LIN {X 0,Y 525.332,Z 477.044,A -85,B 0,C 180,E1 -4784.626,E2 -4784.626} C_VEL
LIN {X 0,Y 525.652,Z 463.482,A -85,B 0,C 180,E1 -4785.311,E2 -4785.311} C_VEL
LIN {X 0,Y 525.936,Z 448.87,A -85,B 0,C 180,E1 -4785.862,E2 -4785.862} C_VEL
LIN {X 0,Y 526.206,Z 434.89,A -85,B 0,C 180,E1 -4786.225,E2 -4786.225} C_VEL
LIN {X 0,Y 526.347,Z 409.491,A -85,B 0,C 180,E1 -4786.608,E2 -4786.608} C_VEL
LIN {X 0,Y 526.914,Z 305.92,A -85,B 0,C 180,E1 -4788.059,E2 -4788.059} C_VEL
LIN {X 0,Y 525.207,Z 295.454,A -85,B 0,C 180,E1 -4788.29,E2 -4788.29} C_VEL
LIN {X 0,Y 525.997,Z 269.747,A -85,B 0,C 180,E1 -4791.557,E2 -4791.557} C_VEL
LIN {X 0,Y 526.502,Z 253.973,A -85,B 0,C 180,E1 -4793.606,E2 -4793.606} C_VEL
LIN {X 0,Y 524.008,Z 242.955,A -85,B 0,C 180,E1 -4795.243,E2 -4795.243} C_VEL
LIN {X 0,Y 523.969,Z 242.84,A -85,B 0,C 180,E1 -4797.998,E2 -4797.998} C_VEL
LIN {X 0,Y 523.943,Z 242.842,A -85,B 0,C 180,E1 -4800.854,E2 -4800.854} C_VEL
LIN {X 0,Y 523.957,Z 242.841,A -85,B 0,C 180,E1 -4803.734,E2 -4803.734} C_VEL
LIN {X 0,Y 523.9,Z 242.841,A -85,B 0,C 180,E1 -4806.401,E2 -4806.401} C_VEL
LIN {X 0,Y 523.917,Z 242.846,A -85,B 0,C 180,E1 -4809.084,E2 -4809.084} C_VEL
LIN {X 0,Y 523.952,Z 242.844,A -85,B 0,C 180,E1 -4812.118,E2 -4812.118} C_VEL
LIN {X 0,Y 523.951,Z 242.838,A -85,B 0,C 180,E1 -4815.308,E2 -4815.308} C_VEL
LIN {X 0,Y 523.957,Z 242.838,A -85,B 0,C 180,E1 -4818.689,E2 -4818.689} C_VEL
LIN {X 0,Y 523.912,Z 242.85,A -85,B 0,C 180,E1 -4821.898,E2 -4821.898} C_VEL
LIN {X 0,Y 523.933,Z 242.839,A -85,B 0,C 180,E1 -4824.908,E2 -4824.908} C_VEL
LIN {X 0,Y 523.937,Z 242.845,A -85,B 0,C 180,E1 -4827.678,E2 -4827.678} C_VEL
LIN {X 0,Y 523.957,Z 242.834,A -85,B 0,C 180,E1 -4830.674,E2 -4830.674} C_VEL
LIN {X 0,Y 523.969,Z 242.843,A -85,B 0,C 180,E1 -4833.728,E2 -4833.728} C_VEL
LIN {X 0,Y 523.93,Z 242.846,A -85,B 0,C 180,E1 -4836.271,E2 -4836.271} C_VEL
LIN {X 0,Y 523.939,Z 242.84,A -85,B 0,C 180,E1 -4838.767,E2 -4838.767} C_VEL
LIN {X 0,Y 523.947,Z 242.841,A -85,B 0,C 180,E1 -4841.221,E2 -4841.221} C_VEL
LIN {X 0,Y 523.934,Z 242.847,A -85,B 0,C 180,E1 -4843.639,E2 -4843.639} C_VEL
LIN {X 0,Y 523.934,Z 242.846,A -85,B 0,C 180,E1 -4846.028,E2 -4846.028} C_VEL
LIN {X 0,Y 524.005,Z 242.832,A -85,B 0,C 180,E1 -4848.394,E2 -4848.394} C_VEL
LIN {X 0,Y 523.999,Z 242.84,A -85,B 0,C 180,E1 -4851.516,E2 -4851.516} C_VEL
LIN {X 0,Y 524.077,Z 242.824,A -85,B 0,C 180,E1 -4854.614,E2 -4854.614} C_VEL
LIN {X 0,Y 524.105,Z 242.826,A -85,B 0,C 180,E1 -4857.695,E2 -4857.695} C_VEL
LIN {X 0,Y 524.118,Z 242.819,A -85,B 0,C 180,E1 -4860.769,E2 -4860.769} C_VEL
LIN {X 0,Y 524.068,Z 242.825,A -85,B 0,C 180,E1 -4863.075,E2 -4863.075} C_VEL
LIN {X 0,Y 524.04,Z 242.827,A -85,B 0,C 180,E1 -4866.159,E2 -4866.159} C_VEL
LIN {X 0,Y 523.994,Z 242.841,A -85,B 0,C 180,E1 -4869.262,E2 -4869.262} C_VEL
LIN {X 0,Y 523.996,Z 242.836,A -85,B 0,C 180,E1 -4871.74,E2 -4871.74} C_VEL
LIN {X 0,Y 523.987,Z 242.84,A -85,B 0,C 180,E1 -4875.053,E2 -4875.053} C_VEL
LIN {X 0,Y 523.959,Z 242.84,A -85,B 0,C 180,E1 -4877.97,E2 -4877.97} C_VEL
LIN {X 0,Y 523.967,Z 242.836,A -85,B 0,C 180,E1 -4880.411,E2 -4880.411} C_VEL
LIN {X 0,Y 523.912,Z 242.85,A -85,B 0,C 180,E1 -4882.894,E2 -4882.894} C_VEL
LIN {X 0,Y 523.948,Z 242.845,A -85,B 0,C 180,E1 -4885.419,E2 -4885.419} C_VEL
LIN {X 0,Y 523.966,Z 242.833,A -85,B 0,C 180,E1 -4888,E2 -4888} C_VEL
LIN {X 0,Y 523.944,Z 242.843,A -85,B 0,C 180,E1 -4890.856,E2 -4890.856} C_VEL
LIN {X 0,Y 523.958,Z 242.837,A -85,B 0,C 180,E1 -4893.736,E2 -4893.736} C_VEL
LIN {X 0,Y 523.92,Z 242.843,A -85,B 0,C 180,E1 -4896.405,E2 -4896.405} C_VEL
LIN {X 0,Y 523.921,Z 242.845,A -85,B 0,C 180,E1 -4899.085,E2 -4899.085} C_VEL
LIN {X 0,Y 523.952,Z 242.841,A -85,B 0,C 180,E1 -4902.12,E2 -4902.12} C_VEL
LIN {X 0,Y 523.955,Z 242.843,A -85,B 0,C 180,E1 -4905.309,E2 -4905.309} C_VEL
LIN {X 0,Y 523.923,Z 242.847,A -85,B 0,C 180,E1 -4906.918,E2 -4906.918} C_VEL
LIN {X 0,Y 523.256,Z 242.926,A -85,B 0,C 180,E1 -4907.56,E2 -4907.56} C_VEL
LIN {X 0,Y 520.412,Z 243.286,A -85,B 0,C 180,E1 -4908.601,E2 -4908.601} C_VEL
LIN {X 0,Y 518.006,Z 243.59,A -85,B 0,C 180,E1 -4909.44,E2 -4909.44} C_VEL
LIN {X 0,Y 516.968,Z 243.716,A -85,B 0,C 180,E1 -4910.088,E2 -4910.088} C_VEL
LIN {X 0,Y 516.881,Z 243.723,A -85,B 0,C 180,E1 -4910.307,E2 -4910.307} C_VEL
LIN {X 0,Y 516.878,Z 243.724,A -85,B 0,C 180,E1 -4913.344,E2 -4913.344} C_VEL
LIN {X 0,Y 516.886,Z 243.716,A -85,B 0,C 180,E1 -4916.12,E2 -4916.12} C_VEL
LIN {X 0,Y 516.892,Z 243.717,A -85,B 0,C 180,E1 -4918.937,E2 -4918.937} C_VEL
LIN {X 0,Y 516.943,Z 243.918,A -85,B 0,C 180,E1 -4921.799,E2 -4921.799} C_VEL
LIN {X 0,Y 519.069,Z 253.792,A -85,B 0,C 180,E1 -4923.461,E2 -4923.461} C_VEL
LIN {X 0,Y 519.119,Z 260.818,A -85,B 0,C 180,E1 -4924.543,E2 -4924.543} C_VEL
LIN {X 0,Y 518.393,Z 281.839,A -85,B 0,C 180,E1 -4927.691,E2 -4927.691} C_VEL
LIN {X 0,Y 517.797,Z 304.258,A -85,B 0,C 180,E1 -4930.989,E2 -4930.989} C_VEL
LIN {X 0,Y 517.551,Z 314.996,A -85,B 0,C 180,E1 -4932.528,E2 -4932.528} C_VEL
LIN {X 0,Y 519.391,Z 327.308,A -85,B 0,C 180,E1 -4932.783,E2 -4932.783} C_VEL
LIN {X 0,Y 519.012,Z 424.803,A -85,B 0,C 180,E1 -4934.123,E2 -4934.123} C_VEL
LIN {X 0,Y 518.798,Z 437.066,A -85,B 0,C 180,E1 -4934.432,E2 -4934.432} C_VEL
LIN {X 0,Y 518.519,Z 450.121,A -85,B 0,C 180,E1 -4934.926,E2 -4934.926} C_VEL
LIN {X 0,Y 518.167,Z 462.487,A -85,B 0,C 180,E1 -4935.569,E2 -4935.569} C_VEL
LIN {X 0,Y 517.756,Z 474.085,A -85,B 0,C 180,E1 -4936.359,E2 -4936.359} C_VEL
LIN {X 0,Y 517.433,Z 484.503,A -85,B 0,C 180,E1 -4937.249,E2 -4937.249} C_VEL
LIN {X 0,Y 517.067,Z 493.894,A -85,B 0,C 180,E1 -4938.236,E2 -4938.236} C_VEL
LIN {X 0,Y 516.846,Z 502.93,A -85,B 0,C 180,E1 -4939.422,E2 -4939.422} C_VEL
LIN {X 0,Y 516.651,Z 510.21,A -85,B 0,C 180,E1 -4940.605,E2 -4940.605} C_VEL
LIN {X 0,Y 516.474,Z 516.049,A -85,B 0,C 180,E1 -4941.786,E2 -4941.786} C_VEL
LIN {X 0,Y 516.398,Z 520.658,A -85,B 0,C 180,E1 -4942.964,E2 -4942.964} C_VEL
LIN {X 0,Y 516.311,Z 523.127,A -85,B 0,C 180,E1 -4943.748,E2 -4943.748} C_VEL
LIN {X 0,Y 516.318,Z 525.122,A -85,B 0,C 180,E1 -4944.532,E2 -4944.532} C_VEL
LIN {X 0,Y 516.227,Z 526.71,A -85,B 0,C 180,E1 -4945.315,E2 -4945.315} C_VEL
LIN {X 0,Y 516.325,Z 527.898,A -85,B 0,C 180,E1 -4946.098,E2 -4946.098} C_VEL
LIN {X 0,Y 516.26,Z 529.038,A -85,B 0,C 180,E1 -4947.659,E2 -4947.659} C_VEL
LIN {X 0,Y 516.161,Z 528.663,A -85,B 0,C 180,E1 -4949.22,E2 -4949.22} C_VEL
LIN {X 0,Y 516.162,Z 527.89,A -85,B 0,C 180,E1 -4950,E2 -4950} C_VEL
LIN {X 0,Y 516.222,Z 525.112,A -85,B 0,C 180,E1 -4951.56,E2 -4951.56} C_VEL
LIN {X 0,Y 516.347,Z 521.938,A -85,B 0,C 180,E1 -4952.73,E2 -4952.73} C_VEL
LIN {X 0,Y 516.43,Z 517.732,A -85,B 0,C 180,E1 -4953.902,E2 -4953.902} C_VEL
LIN {X 0,Y 516.636,Z 512.373,A -85,B 0,C 180,E1 -4955.073,E2 -4955.073} C_VEL
LIN {X 0,Y 516.742,Z 505.703,A -85,B 0,C 180,E1 -4956.246,E2 -4956.246} C_VEL
LIN {X 0,Y 517,Z 497.426,A -85,B 0,C 180,E1 -4957.42,E2 -4957.42} C_VEL
LIN {X 0,Y 517.34,Z 488.918,A -85,B 0,C 180,E1 -4958.397,E2 -4958.397} C_VEL
LIN {X 0,Y 517.677,Z 478.474,A -85,B 0,C 180,E1 -4959.376,E2 -4959.376} C_VEL
LIN {X 0,Y 517.974,Z 468.125,A -85,B 0,C 180,E1 -4960.159,E2 -4960.159} C_VEL
LIN {X 0,Y 518.32,Z 456.727,A -85,B 0,C 180,E1 -4960.844,E2 -4960.844} C_VEL
LIN {X 0,Y 518.643,Z 443.643,A -85,B 0,C 180,E1 -4961.43,E2 -4961.43} C_VEL
LIN {X 0,Y 518.865,Z 430.369,A -85,B 0,C 180,E1 -4961.846,E2 -4961.846} C_VEL
LIN {X 0,Y 519.002,Z 417.033,A -85,B 0,C 180,E1 -4962.091,E2 -4962.091} C_VEL
LIN {X 0,Y 519.312,Z 325.809,A -85,B 0,C 180,E1 -4963.329,E2 -4963.329} C_VEL
LIN {X 0,Y 517.579,Z 315.248,A -85,B 0,C 180,E1 -4963.546,E2 -4963.546} C_VEL
LIN {X 0,Y 517.655,Z 309.433,A -85,B 0,C 180,E1 -4964.345,E2 -4964.345} C_VEL
LIN {X 0,Y 518.24,Z 287.488,A -85,B 0,C 180,E1 -4967.562,E2 -4967.562} C_VEL
LIN {X 0,Y 518.798,Z 268.307,A -85,B 0,C 180,E1 -4970.415,E2 -4970.415} C_VEL
LIN {X 0,Y 519.199,Z 254.521,A -85,B 0,C 180,E1 -4972.493,E2 -4972.493} C_VEL
LIN {X 0,Y 516.928,Z 243.789,A -85,B 0,C 180,E1 -4974.295,E2 -4974.295} C_VEL
LIN {X 0,Y 516.926,Z 243.707,A -85,B 0,C 180,E1 -4976.657,E2 -4976.657} C_VEL
LIN {X 0,Y 516.913,Z 243.716,A -85,B 0,C 180,E1 -4979.523,E2 -4979.523} C_VEL
LIN {X 0,Y 516.899,Z 243.718,A -85,B 0,C 180,E1 -4982.543,E2 -4982.543} C_VEL
LIN {X 0,Y 516.867,Z 243.726,A -85,B 0,C 180,E1 -4985.329,E2 -4985.329} C_VEL
LIN {X 0,Y 516.88,Z 243.721,A -85,B 0,C 180,E1 -4987.942,E2 -4987.942} C_VEL
LIN {X 0,Y 516.885,Z 243.721,A -85,B 0,C 180,E1 -4990.741,E2 -4990.741} C_VEL
LIN {X 0,Y 516.905,Z 243.721,A -85,B 0,C 180,E1 -4992.828,E2 -4992.828} C_VEL
LIN {X 0,Y 516.922,Z 243.718,A -85,B 0,C 180,E1 -4995.009,E2 -4995.009} C_VEL
LIN {X 0,Y 516.913,Z 243.717,A -85,B 0,C 180,E1 -4998.398,E2 -4998.398} C_VEL
LIN {X 0,Y 516.881,Z 243.726,A -85,B 0,C 180,E1 -5001.283,E2 -5001.283} C_VEL
LIN {X 0,Y 516.888,Z 243.719,A -85,B 0,C 180,E1 -5004.22,E2 -5004.22} C_VEL
LIN {X 0,Y 516.894,Z 243.718,A -85,B 0,C 180,E1 -5007.052,E2 -5007.052} C_VEL
LIN {X 0,Y 516.897,Z 243.719,A -85,B 0,C 180,E1 -5009.796,E2 -5009.796} C_VEL
LIN {X 0,Y 516.924,Z 243.715,A -85,B 0,C 180,E1 -5012.467,E2 -5012.467} C_VEL
LIN {X 0,Y 516.906,Z 243.72,A -85,B 0,C 180,E1 -5015.071,E2 -5015.071} C_VEL
LIN {X 0,Y 516.864,Z 243.723,A -85,B 0,C 180,E1 -5017.621,E2 -5017.621} C_VEL
LIN {X 0,Y 516.927,Z 243.714,A -85,B 0,C 180,E1 -5020.129,E2 -5020.129} C_VEL
LIN {X 0,Y 516.925,Z 243.721,A -85,B 0,C 180,E1 -5022.596,E2 -5022.596} C_VEL
LIN {X 0,Y 516.935,Z 243.716,A -85,B 0,C 180,E1 -5025.03,E2 -5025.03} C_VEL
LIN {X 0,Y 516.958,Z 243.714,A -85,B 0,C 180,E1 -5028.233,E2 -5028.233} C_VEL
LIN {X 0,Y 516.963,Z 243.71,A -85,B 0,C 180,E1 -5031.399,E2 -5031.399} C_VEL
LIN {X 0,Y 517.003,Z 243.705,A -85,B 0,C 180,E1 -5033.756,E2 -5033.756} C_VEL
LIN {X 0,Y 517.077,Z 243.696,A -85,B 0,C 180,E1 -5037.663,E2 -5037.663} C_VEL
LIN {X 0,Y 517.088,Z 243.697,A -85,B 0,C 180,E1 -5040.779,E2 -5040.779} C_VEL
LIN {X 0,Y 517.008,Z 243.705,A -85,B 0,C 180,E1 -5043.117,E2 -5043.117} C_VEL
LIN {X 0,Y 517.003,Z 243.709,A -85,B 0,C 180,E1 -5046.243,E2 -5046.243} C_VEL
LIN {X 0,Y 516.948,Z 243.712,A -85,B 0,C 180,E1 -5049.389,E2 -5049.389} C_VEL
LIN {X 0,Y 516.944,Z 243.712,A -85,B 0,C 180,E1 -5051.807,E2 -5051.807} C_VEL
LIN {X 0,Y 516.936,Z 243.712,A -85,B 0,C 180,E1 -5055.146,E2 -5055.146} C_VEL
LIN {X 0,Y 516.918,Z 243.724,A -85,B 0,C 180,E1 -5058.222,E2 -5058.222} C_VEL
LIN {X 0,Y 516.905,Z 243.717,A -85,B 0,C 180,E1 -5060.702,E2 -5060.702} C_VEL
LIN {X 0,Y 516.904,Z 243.724,A -85,B 0,C 180,E1 -5064.072,E2 -5064.072} C_VEL
LIN {X 0,Y 516.92,Z 243.717,A -85,B 0,C 180,E1 -5066.658,E2 -5066.658} C_VEL
LIN {X 0,Y 516.918,Z 243.715,A -85,B 0,C 180,E1 -5069.527,E2 -5069.527} C_VEL
LIN {X 0,Y 516.894,Z 243.72,A -85,B 0,C 180,E1 -5072.545,E2 -5072.545} C_VEL
LIN {X 0,Y 516.877,Z 243.722,A -85,B 0,C 180,E1 -5075.333,E2 -5075.333} C_VEL
LIN {X 0,Y 516.877,Z 243.725,A -85,B 0,C 180,E1 -5077.944,E2 -5077.944} C_VEL
LIN {X 0,Y 516.881,Z 243.72,A -85,B 0,C 180,E1 -5080.742,E2 -5080.742} C_VEL
LIN {X 0,Y 516.879,Z 243.718,A -85,B 0,C 180,E1 -5082.832,E2 -5082.832} C_VEL
LIN {X 0,Y 516.918,Z 243.717,A -85,B 0,C 180,E1 -5085.011,E2 -5085.011} C_VEL
LIN {X 0,Y 516.912,Z 243.705,A -85,B 0,C 180,E1 -5088.399,E2 -5088.399} C_VEL
LIN {X 0,Y 516.877,Z 243.725,A -85,B 0,C 180,E1 -5091.285,E2 -5091.285} C_VEL
LIN {X 0,Y 516.868,Z 243.716,A -85,B 0,C 180,E1 -5094.22,E2 -5094.22} C_VEL
LIN {X 0,Y 516.894,Z 243.723,A -85,B 0,C 180,E1 -5097.054,E2 -5097.054} C_VEL
LIN {X 0,Y 516.891,Z 243.726,A -85,B 0,C 180,E1 -5099.797,E2 -5099.797} C_VEL
LIN {X 0,Y 516.927,Z 243.719,A -85,B 0,C 180,E1 -5102.468,E2 -5102.468} C_VEL
LIN {X 0,Y 516.958,Z 243.855,A -85,B 0,C 180,E1 -5104.537,E2 -5104.537} C_VEL
LIN {X 0,Y 519.629,Z 255.55,A -85,B 0,C 180,E1 -5106.274,E2 -5106.274} C_VEL
LIN {X 0,Y 519.014,Z 274.477,A -85,B 0,C 180,E1 -5108.761,E2 -5108.761} C_VEL
LIN {X 0,Y 518.331,Z 295.82,A -85,B 0,C 180,E1 -5111.495,E2 -5111.495} C_VEL
LIN {X 0,Y 520.162,Z 307.48,A -85,B 0,C 180,E1 -5111.741,E2 -5111.741} C_VEL
LIN {X 0,Y 519.337,Z 432.731,A -85,B 0,C 180,E1 -5113.537,E2 -5113.537} C_VEL
LIN {X 0,Y 519.113,Z 447.385,A -85,B 0,C 180,E1 -5113.905,E2 -5113.905} C_VEL
LIN {X 0,Y 518.835,Z 460.485,A -85,B 0,C 180,E1 -5114.382,E2 -5114.382} C_VEL
LIN {X 0,Y 518.488,Z 472.87,A -85,B 0,C 180,E1 -5114.976,E2 -5114.976} C_VEL
LIN {X 0,Y 518.09,Z 485.849,A -85,B 0,C 180,E1 -5115.767,E2 -5115.767} C_VEL
LIN {X 0,Y 517.703,Z 497.626,A -85,B 0,C 180,E1 -5116.657,E2 -5116.657} C_VEL
LIN {X 0,Y 517.381,Z 508.456,A -85,B 0,C 180,E1 -5117.652,E2 -5117.652} C_VEL
LIN {X 0,Y 517.067,Z 519.064,A -85,B 0,C 180,E1 -5118.832,E2 -5118.832} C_VEL
LIN {X 0,Y 516.798,Z 527.848,A -85,B 0,C 180,E1 -5120.015,E2 -5120.015} C_VEL
LIN {X 0,Y 516.579,Z 536.259,A -85,B 0,C 180,E1 -5121.393,E2 -5121.393} C_VEL
LIN {X 0,Y 516.445,Z 542.107,A -85,B 0,C 180,E1 -5122.572,E2 -5122.572} C_VEL
LIN {X 0,Y 516.371,Z 546.91,A -85,B 0,C 180,E1 -5123.749,E2 -5123.749} C_VEL
LIN {X 0,Y 516.305,Z 550.799,A -85,B 0,C 180,E1 -5124.924,E2 -5124.924} C_VEL
LIN {X 0,Y 516.324,Z 553.783,A -85,B 0,C 180,E1 -5126.098,E2 -5126.098} C_VEL
LIN {X 0,Y 516.259,Z 556.518,A -85,B 0,C 180,E1 -5127.659,E2 -5127.659} C_VEL
LIN {X 0,Y 516.157,Z 557.872,A -85,B 0,C 180,E1 -5129.22,E2 -5129.22} C_VEL
LIN {X 0,Y 516.157,Z 557.873,A -85,B 0,C 180,E1 -5130.78,E2 -5130.78} C_VEL
LIN {X 0,Y 516.259,Z 556.521,A -85,B 0,C 180,E1 -5132.341,E2 -5132.341} C_VEL
LIN {X 0,Y 516.324,Z 553.788,A -85,B 0,C 180,E1 -5133.902,E2 -5133.902} C_VEL
LIN {X 0,Y 516.361,Z 549.595,A -85,B 0,C 180,E1 -5135.467,E2 -5135.467} C_VEL
LIN {X 0,Y 516.401,Z 543.811,A -85,B 0,C 180,E1 -5137.036,E2 -5137.036} C_VEL
LIN {X 0,Y 516.576,Z 537.283,A -85,B 0,C 180,E1 -5138.41,E2 -5138.41} C_VEL
LIN {X 0,Y 516.755,Z 529.161,A -85,B 0,C 180,E1 -5139.788,E2 -5139.788} C_VEL
LIN {X 0,Y 517.024,Z 520.647,A -85,B 0,C 180,E1 -5140.97,E2 -5140.97} C_VEL
LIN {X 0,Y 517.356,Z 510.186,A -85,B 0,C 180,E1 -5142.173,E2 -5142.173} C_VEL
LIN {X 0,Y 517.686,Z 498.799,A -85,B 0,C 180,E1 -5143.243,E2 -5143.243} C_VEL
LIN {X 0,Y 518.041,Z 487.272,A -85,B 0,C 180,E1 -5144.134,E2 -5144.134} C_VEL
LIN {X 0,Y 518.454,Z 474.626,A -85,B 0,C 180,E1 -5144.925,E2 -5144.925} C_VEL
LIN {X 0,Y 518.836,Z 461.58,A -85,B 0,C 180,E1 -5145.567,E2 -5145.567} C_VEL
LIN {X 0,Y 519.11,Z 447.456,A -85,B 0,C 180,E1 -5146.091,E2 -5146.091} C_VEL
LIN {X 0,Y 519.357,Z 433.721,A -85,B 0,C 180,E1 -5146.44,E2 -5146.44} C_VEL
LIN {X 0,Y 520.139,Z 307.017,A -85,B 0,C 180,E1 -5148.266,E2 -5148.266} C_VEL
LIN {X 0,Y 518.335,Z 295.775,A -85,B 0,C 180,E1 -5148.507,E2 -5148.507} C_VEL
LIN {X 0,Y 519.165,Z 269.763,A -85,B 0,C 180,E1 -5151.855,E2 -5151.855} C_VEL
LIN {X 0,Y 519.644,Z 255.59,A -85,B 0,C 180,E1 -5153.725,E2 -5153.725} C_VEL
LIN {X 0,Y 516.969,Z 243.829,A -85,B 0,C 180,E1 -5155.503,E2 -5155.503} C_VEL
LIN {X 0,Y 516.918,Z 243.714,A -85,B 0,C 180,E1 -5158.415,E2 -5158.415} C_VEL
LIN {X 0,Y 516.888,Z 243.718,A -85,B 0,C 180,E1 -5161.109,E2 -5161.109} C_VEL
LIN {X 0,Y 516.906,Z 243.721,A -85,B 0,C 180,E1 -5163.966,E2 -5163.966} C_VEL
LIN {X 0,Y 516.874,Z 243.716,A -85,B 0,C 180,E1 -5166.746,E2 -5166.746} C_VEL
LIN {X 0,Y 516.879,Z 243.723,A -85,B 0,C 180,E1 -5169.721,E2 -5169.721} C_VEL
LIN {X 0,Y 516.903,Z 243.721,A -85,B 0,C 180,E1 -5172.76,E2 -5172.76} C_VEL
LIN {X 0,Y 516.919,Z 243.715,A -85,B 0,C 180,E1 -5175.01,E2 -5175.01} C_VEL
LIN {X 0,Y 516.913,Z 243.717,A -85,B 0,C 180,E1 -5178.398,E2 -5178.398} C_VEL
LIN {X 0,Y 516.878,Z 243.722,A -85,B 0,C 180,E1 -5181.284,E2 -5181.284} C_VEL
LIN {X 0,Y 516.886,Z 243.72,A -85,B 0,C 180,E1 -5184.221,E2 -5184.221} C_VEL
LIN {X 0,Y 516.892,Z 243.719,A -85,B 0,C 180,E1 -5187.053,E2 -5187.053} C_VEL
LIN {X 0,Y 516.895,Z 243.718,A -85,B 0,C 180,E1 -5189.797,E2 -5189.797} C_VEL
LIN {X 0,Y 516.923,Z 243.718,A -85,B 0,C 180,E1 -5192.467,E2 -5192.467} C_VEL
LIN {X 0,Y 516.904,Z 243.717,A -85,B 0,C 180,E1 -5195.072,E2 -5195.072} C_VEL
LIN {X 0,Y 516.863,Z 243.727,A -85,B 0,C 180,E1 -5197.621,E2 -5197.621} C_VEL
LIN {X 0,Y 516.925,Z 243.72,A -85,B 0,C 180,E1 -5200.13,E2 -5200.13} C_VEL
LIN {X 0,Y 516.925,Z 243.714,A -85,B 0,C 180,E1 -5202.596,E2 -5202.596} C_VEL
LIN {X 0,Y 516.935,Z 243.713,A -85,B 0,C 180,E1 -5205.03,E2 -5205.03} C_VEL
LIN {X 0,Y 516.958,Z 243.711,A -85,B 0,C 180,E1 -5208.234,E2 -5208.234} C_VEL
LIN {X 0,Y 516.963,Z 243.715,A -85,B 0,C 180,E1 -5211.4,E2 -5211.4} C_VEL
LIN {X 0,Y 517.004,Z 243.712,A -85,B 0,C 180,E1 -5213.757,E2 -5213.757} C_VEL
LIN {X 0,Y 517.077,Z 243.701,A -85,B 0,C 180,E1 -5217.663,E2 -5217.663} C_VEL
LIN {X 0,Y 517.088,Z 243.695,A -85,B 0,C 180,E1 -5220.779,E2 -5220.779} C_VEL
LIN {X 0,Y 517.009,Z 243.705,A -85,B 0,C 180,E1 -5223.117,E2 -5223.117} C_VEL
LIN {X 0,Y 517.004,Z 243.703,A -85,B 0,C 180,E1 -5226.244,E2 -5226.244} C_VEL
LIN {X 0,Y 516.948,Z 243.721,A -85,B 0,C 180,E1 -5229.39,E2 -5229.39} C_VEL
LIN {X 0,Y 516.946,Z 243.714,A -85,B 0,C 180,E1 -5231.808,E2 -5231.808} C_VEL
LIN {X 0,Y 516.938,Z 243.72,A -85,B 0,C 180,E1 -5235.147,E2 -5235.147} C_VEL
LIN {X 0,Y 516.921,Z 243.716,A -85,B 0,C 180,E1 -5238.223,E2 -5238.223} C_VEL
LIN {X 0,Y 516.907,Z 243.717,A -85,B 0,C 180,E1 -5240.702,E2 -5240.702} C_VEL
LIN {X 0,Y 516.907,Z 243.716,A -85,B 0,C 180,E1 -5244.073,E2 -5244.073} C_VEL
LIN {X 0,Y 516.922,Z 243.719,A -85,B 0,C 180,E1 -5246.658,E2 -5246.658} C_VEL
LIN {X 0,Y 516.907,Z 243.716,A -85,B 0,C 180,E1 -5249.525,E2 -5249.525} C_VEL
LIN {X 0,Y 516.897,Z 243.722,A -85,B 0,C 180,E1 -5252.545,E2 -5252.545} C_VEL
LIN {X 0,Y 516.88,Z 243.721,A -85,B 0,C 180,E1 -5255.333,E2 -5255.333} C_VEL
LIN {X 0,Y 516.88,Z 243.721,A -85,B 0,C 180,E1 -5257.944,E2 -5257.944} C_VEL
LIN {X 0,Y 516.883,Z 243.721,A -85,B 0,C 180,E1 -5260.742,E2 -5260.742} C_VEL
LIN {X 0,Y 516.881,Z 243.727,A -85,B 0,C 180,E1 -5262.832,E2 -5262.832} C_VEL
LIN {X 0,Y 516.922,Z 243.723,A -85,B 0,C 180,E1 -5265.011,E2 -5265.011} C_VEL
LIN {X 0,Y 516.917,Z 243.718,A -85,B 0,C 180,E1 -5268.399,E2 -5268.399} C_VEL
LIN {X 0,Y 516.881,Z 243.723,A -85,B 0,C 180,E1 -5270.307,E2 -5270.307} C_VEL
LIN {X 0,Y 516.21,Z 243.799,A -85,B 0,C 180,E1 -5270.957,E2 -5270.957} C_VEL
LIN {X 0,Y 513.363,Z 244.153,A -85,B 0,C 180,E1 -5272.013,E2 -5272.013} C_VEL
LIN {X 0,Y 510.954,Z 244.458,A -85,B 0,C 180,E1 -5272.863,E2 -5272.863} C_VEL
LIN {X 0,Y 509.91,Z 244.592,A -85,B 0,C 180,E1 -5273.52,E2 -5273.52} C_VEL
LIN {X 0,Y 509.821,Z 244.602,A -85,B 0,C 180,E1 -5273.742,E2 -5273.742} C_VEL
LIN {X 0,Y 509.843,Z 244.595,A -85,B 0,C 180,E1 -5276.539,E2 -5276.539} C_VEL
LIN {X 0,Y 509.845,Z 244.594,A -85,B 0,C 180,E1 -5279.335,E2 -5279.335} C_VEL
LIN {X 0,Y 509.896,Z 244.829,A -85,B 0,C 180,E1 -5281.554,E2 -5281.554} C_VEL
LIN {X 0,Y 512.355,Z 256.555,A -85,B 0,C 180,E1 -5283.547,E2 -5283.547} C_VEL
LIN {X 0,Y 511.831,Z 273.246,A -85,B 0,C 180,E1 -5286.105,E2 -5286.105} C_VEL
LIN {X 0,Y 511.197,Z 291.439,A -85,B 0,C 180,E1 -5288.846,E2 -5288.846} C_VEL
LIN {X 0,Y 510.636,Z 313.126,A -85,B 0,C 180,E1 -5292.062,E2 -5292.062} C_VEL
LIN {X 0,Y 510.626,Z 315.286,A -85,B 0,C 180,E1 -5292.311,E2 -5292.311} C_VEL
LIN {X 0,Y 512.602,Z 327.693,A -85,B 0,C 180,E1 -5292.561,E2 -5292.561} C_VEL
LIN {X 0,Y 512.185,Z 425.03,A -85,B 0,C 180,E1 -5293.905,E2 -5293.905} C_VEL
LIN {X 0,Y 511.977,Z 437.286,A -85,B 0,C 180,E1 -5294.219,E2 -5294.219} C_VEL
LIN {X 0,Y 511.67,Z 450.338,A -85,B 0,C 180,E1 -5294.72,E2 -5294.72} C_VEL
LIN {X 0,Y 511.311,Z 462.689,A -85,B 0,C 180,E1 -5295.371,E2 -5295.371} C_VEL
LIN {X 0,Y 510.846,Z 474.274,A -85,B 0,C 180,E1 -5296.17,E2 -5296.17} C_VEL
LIN {X 0,Y 510.511,Z 484.677,A -85,B 0,C 180,E1 -5297.073,E2 -5297.073} C_VEL
LIN {X 0,Y 510.093,Z 494.057,A -85,B 0,C 180,E1 -5298.073,E2 -5298.073} C_VEL
LIN {X 0,Y 509.845,Z 503.082,A -85,B 0,C 180,E1 -5299.275,E2 -5299.275} C_VEL
LIN {X 0,Y 509.592,Z 510.357,A -85,B 0,C 180,E1 -5300.474,E2 -5300.474} C_VEL
LIN {X 0,Y 509.433,Z 516.195,A -85,B 0,C 180,E1 -5301.671,E2 -5301.671} C_VEL
LIN {X 0,Y 509.323,Z 520.807,A -85,B 0,C 180,E1 -5302.866,E2 -5302.866} C_VEL
LIN {X 0,Y 509.262,Z 523.284,A -85,B 0,C 180,E1 -5303.662,E2 -5303.662} C_VEL
LIN {X 0,Y 509.248,Z 525.282,A -85,B 0,C 180,E1 -5304.456,E2 -5304.456} C_VEL
LIN {X 0,Y 509.145,Z 526.873,A -85,B 0,C 180,E1 -5305.249,E2 -5305.249} C_VEL
LIN {X 0,Y 509.232,Z 528.068,A -85,B 0,C 180,E1 -5306.043,E2 -5306.043} C_VEL
LIN {X 0,Y 509.192,Z 528.851,A -85,B 0,C 180,E1 -5306.835,E2 -5306.835} C_VEL
LIN {X 0,Y 509.189,Z 529.232,A -85,B 0,C 180,E1 -5307.627,E2 -5307.627} C_VEL
LIN {X 0,Y 509.075,Z 528.879,A -85,B 0,C 180,E1 -5309.209,E2 -5309.209} C_VEL
LIN {X 0,Y 509.073,Z 528.132,A -85,B 0,C 180,E1 -5310,E2 -5310} C_VEL
LIN {X 0,Y 509.141,Z 525.393,A -85,B 0,C 180,E1 -5311.582,E2 -5311.582} C_VEL
LIN {X 0,Y 509.279,Z 522.259,A -85,B 0,C 180,E1 -5312.768,E2 -5312.768} C_VEL
LIN {X 0,Y 509.365,Z 518.101,A -85,B 0,C 180,E1 -5313.956,E2 -5313.956} C_VEL
LIN {X 0,Y 509.584,Z 512.795,A -85,B 0,C 180,E1 -5315.143,E2 -5315.143} C_VEL
LIN {X 0,Y 509.712,Z 506.187,A -85,B 0,C 180,E1 -5316.333,E2 -5316.333} C_VEL
LIN {X 0,Y 510.006,Z 498.007,A -85,B 0,C 180,E1 -5317.522,E2 -5317.522} C_VEL
LIN {X 0,Y 510.371,Z 489.61,A -85,B 0,C 180,E1 -5318.513,E2 -5318.513} C_VEL
LIN {X 0,Y 510.72,Z 479.287,A -85,B 0,C 180,E1 -5319.505,E2 -5319.505} C_VEL
LIN {X 0,Y 511.036,Z 469.088,A -85,B 0,C 180,E1 -5320.299,E2 -5320.299} C_VEL
LIN {X 0,Y 511.433,Z 457.918,A -85,B 0,C 180,E1 -5320.991,E2 -5320.991} C_VEL
LIN {X 0,Y 511.782,Z 445.271,A -85,B 0,C 180,E1 -5321.586,E2 -5321.586} C_VEL
LIN {X 0,Y 512.025,Z 432.591,A -85,B 0,C 180,E1 -5322.007,E2 -5322.007} C_VEL
LIN {X 0,Y 512.222,Z 419.353,A -85,B 0,C 180,E1 -5322.279,E2 -5322.279} C_VEL
LIN {X 0,Y 512.517,Z 326.659,A -85,B 0,C 180,E1 -5323.545,E2 -5323.545} C_VEL
LIN {X 0,Y 510.619,Z 315.15,A -85,B 0,C 180,E1 -5323.785,E2 -5323.785} C_VEL
LIN {X 0,Y 510.64,Z 312.372,A -85,B 0,C 180,E1 -5324.14,E2 -5324.14} C_VEL
LIN {X 0,Y 511.182,Z 291.77,A -85,B 0,C 180,E1 -5327.193,E2 -5327.193} C_VEL
LIN {X 0,Y 511.816,Z 272.561,A -85,B 0,C 180,E1 -5330.077,E2 -5330.077} C_VEL
LIN {X 0,Y 512.311,Z 256.088,A -85,B 0,C 180,E1 -5332.588,E2 -5332.588} C_VEL
LIN {X 0,Y 509.851,Z 244.682,A -85,B 0,C 180,E1 -5334.525,E2 -5334.525} C_VEL
LIN {X 0,Y 509.885,Z 244.586,A -85,B 0,C 180,E1 -5337.055,E2 -5337.055} C_VEL
LIN {X 0,Y 509.86,Z 244.593,A -85,B 0,C 180,E1 -5339.75,E2 -5339.75} C_VEL
LIN {X 0,Y 509.876,Z 244.595,A -85,B 0,C 180,E1 -5342.774,E2 -5342.774} C_VEL
LIN {X 0,Y 509.827,Z 244.607,A -85,B 0,C 180,E1 -5345.578,E2 -5345.578} C_VEL
LIN {X 0,Y 509.849,Z 244.596,A -85,B 0,C 180,E1 -5348.337,E2 -5348.337} C_VEL
LIN {X 0,Y 509.858,Z 244.6,A -85,B 0,C 180,E1 -5351.424,E2 -5351.424} C_VEL
LIN {X 0,Y 509.856,Z 244.596,A -85,B 0,C 180,E1 -5354.667,E2 -5354.667} C_VEL
LIN {X 0,Y 509.855,Z 244.596,A -85,B 0,C 180,E1 -5358.102,E2 -5358.102} C_VEL
LIN {X 0,Y 509.845,Z 244.592,A -85,B 0,C 180,E1 -5360.647,E2 -5360.647} C_VEL
LIN {X 0,Y 509.833,Z 244.6,A -85,B 0,C 180,E1 -5363.647,E2 -5363.647} C_VEL
LIN {X 0,Y 509.859,Z 244.589,A -85,B 0,C 180,E1 -5366.539,E2 -5366.539} C_VEL
LIN {X 0,Y 509.847,Z 244.601,A -85,B 0,C 180,E1 -5369.334,E2 -5369.334} C_VEL
LIN {X 0,Y 509.89,Z 244.589,A -85,B 0,C 180,E1 -5372.054,E2 -5372.054} C_VEL
LIN {X 0,Y 509.872,Z 244.6,A -85,B 0,C 180,E1 -5374.703,E2 -5374.703} C_VEL
LIN {X 0,Y 509.822,Z 244.601,A -85,B 0,C 180,E1 -5377.457,E2 -5377.457} C_VEL
LIN {X 0,Y 509.911,Z 244.586,A -85,B 0,C 180,E1 -5379.844,E2 -5379.844} C_VEL
LIN {X 0,Y 509.881,Z 244.595,A -85,B 0,C 180,E1 -5383.174,E2 -5383.174} C_VEL
LIN {X 0,Y 509.858,Z 244.593,A -85,B 0,C 180,E1 -5385.634,E2 -5385.634} C_VEL
LIN {X 0,Y 509.895,Z 244.593,A -85,B 0,C 180,E1 -5388.123,E2 -5388.123} C_VEL
LIN {X 0,Y 509.91,Z 244.589,A -85,B 0,C 180,E1 -5391.279,E2 -5391.279} C_VEL
LIN {X 0,Y 509.972,Z 244.581,A -85,B 0,C 180,E1 -5393.67,E2 -5393.67} C_VEL
LIN {X 0,Y 510.048,Z 244.572,A -85,B 0,C 180,E1 -5397.631,E2 -5397.631} C_VEL
LIN {X 0,Y 510.058,Z 244.572,A -85,B 0,C 180,E1 -5400.789,E2 -5400.789} C_VEL
LIN {X 0,Y 509.95,Z 244.584,A -85,B 0,C 180,E1 -5403.16,E2 -5403.16} C_VEL
LIN {X 0,Y 509.971,Z 244.585,A -85,B 0,C 180,E1 -5406.329,E2 -5406.329} C_VEL
LIN {X 0,Y 509.909,Z 244.592,A -85,B 0,C 180,E1 -5408.72,E2 -5408.72} C_VEL
LIN {X 0,Y 509.896,Z 244.591,A -85,B 0,C 180,E1 -5411.932,E2 -5411.932} C_VEL
LIN {X 0,Y 509.886,Z 244.59,A -85,B 0,C 180,E1 -5415.242,E2 -5415.242} C_VEL
LIN {X 0,Y 509.881,Z 244.598,A -85,B 0,C 180,E1 -5418.001,E2 -5418.001} C_VEL
LIN {X 0,Y 509.843,Z 244.595,A -85,B 0,C 180,E1 -5421.002,E2 -5421.002} C_VEL
LIN {X 0,Y 509.83,Z 244.601,A -85,B 0,C 180,E1 -5423.563,E2 -5423.563} C_VEL
LIN {X 0,Y 509.905,Z 244.594,A -85,B 0,C 180,E1 -5426.379,E2 -5426.379} C_VEL
LIN {X 0,Y 509.879,Z 244.589,A -85,B 0,C 180,E1 -5428.844,E2 -5428.844} C_VEL
LIN {X 0,Y 509.82,Z 244.596,A -85,B 0,C 180,E1 -5431.59,E2 -5431.59} C_VEL
LIN {X 0,Y 509.848,Z 244.599,A -85,B 0,C 180,E1 -5434.414,E2 -5434.414} C_VEL
LIN {X 0,Y 509.814,Z 244.595,A -85,B 0,C 180,E1 -5437.341,E2 -5437.341} C_VEL
LIN {X 0,Y 509.834,Z 244.6,A -85,B 0,C 180,E1 -5440.383,E2 -5440.383} C_VEL
LIN {X 0,Y 509.819,Z 244.598,A -85,B 0,C 180,E1 -5443.063,E2 -5443.063} C_VEL
LIN {X 0,Y 509.827,Z 244.6,A -85,B 0,C 180,E1 -5445.793,E2 -5445.793} C_VEL
LIN {X 0,Y 509.853,Z 244.583,A -85,B 0,C 180,E1 -5448.575,E2 -5448.575} C_VEL
LIN {X 0,Y 509.847,Z 244.602,A -85,B 0,C 180,E1 -5451.787,E2 -5451.787} C_VEL
LIN {X 0,Y 509.827,Z 244.592,A -85,B 0,C 180,E1 -5454.622,E2 -5454.622} C_VEL
LIN {X 0,Y 509.861,Z 244.596,A -85,B 0,C 180,E1 -5457.482,E2 -5457.482} C_VEL
LIN {X 0,Y 509.857,Z 244.598,A -85,B 0,C 180,E1 -5460.274,E2 -5460.274} C_VEL
LIN {X 0,Y 509.884,Z 244.599,A -85,B 0,C 180,E1 -5462.945,E2 -5462.945} C_VEL
LIN {X 0,Y 509.957,Z 244.826,A -85,B 0,C 180,E1 -5464.312,E2 -5464.312} C_VEL
LIN {X 0,Y 512.77,Z 257.109,A -85,B 0,C 180,E1 -5466.152,E2 -5466.152} C_VEL
LIN {X 0,Y 512.104,Z 276.382,A -85,B 0,C 180,E1 -5468.716,E2 -5468.716} C_VEL
LIN {X 0,Y 511.423,Z 295.738,A -85,B 0,C 180,E1 -5471.244,E2 -5471.244} C_VEL
LIN {X 0,Y 513.374,Z 307.942,A -85,B 0,C 180,E1 -5471.518,E2 -5471.518} C_VEL
LIN {X 0,Y 512.481,Z 432.594,A -85,B 0,C 180,E1 -5473.34,E2 -5473.34} C_VEL
LIN {X 0,Y 512.223,Z 446.564,A -85,B 0,C 180,E1 -5473.69,E2 -5473.69} C_VEL
LIN {X 0,Y 511.91,Z 460.8,A -85,B 0,C 180,E1 -5474.217,E2 -5474.217} C_VEL
LIN {X 0,Y 511.505,Z 473.979,A -85,B 0,C 180,E1 -5474.868,E2 -5474.868} C_VEL
LIN {X 0,Y 511.089,Z 486.728,A -85,B 0,C 180,E1 -5475.67,E2 -5475.67} C_VEL
LIN {X 0,Y 510.684,Z 498.337,A -85,B 0,C 180,E1 -5476.572,E2 -5476.572} C_VEL
LIN {X 0,Y 510.341,Z 509.275,A -85,B 0,C 180,E1 -5477.605,E2 -5477.605} C_VEL
LIN {X 0,Y 510.023,Z 518.701,A -85,B 0,C 180,E1 -5478.676,E2 -5478.676} C_VEL
LIN {X 0,Y 509.732,Z 527.523,A -85,B 0,C 180,E1 -5479.875,E2 -5479.875} C_VEL
LIN {X 0,Y 509.526,Z 535.972,A -85,B 0,C 180,E1 -5481.273,E2 -5481.273} C_VEL
LIN {X 0,Y 509.368,Z 541.842,A -85,B 0,C 180,E1 -5482.468,E2 -5482.468} C_VEL
LIN {X 0,Y 509.286,Z 546.667,A -85,B 0,C 180,E1 -5483.662,E2 -5483.662} C_VEL
LIN {X 0,Y 509.234,Z 550.572,A -85,B 0,C 180,E1 -5484.853,E2 -5484.853} C_VEL
LIN {X 0,Y 509.217,Z 553.565,A -85,B 0,C 180,E1 -5486.043,E2 -5486.043} C_VEL
LIN {X 0,Y 509.188,Z 556.313,A -85,B 0,C 180,E1 -5487.627,E2 -5487.627} C_VEL
LIN {X 0,Y 509.071,Z 557.673,A -85,B 0,C 180,E1 -5489.209,E2 -5489.209} C_VEL
LIN {X 0,Y 509.071,Z 557.673,A -85,B 0,C 180,E1 -5490.791,E2 -5490.791} C_VEL
LIN {X 0,Y 509.188,Z 556.315,A -85,B 0,C 180,E1 -5492.373,E2 -5492.373} C_VEL
LIN {X 0,Y 509.217,Z 553.57,A -85,B 0,C 180,E1 -5493.957,E2 -5493.957} C_VEL
LIN {X 0,Y 509.273,Z 549.359,A -85,B 0,C 180,E1 -5495.543,E2 -5495.543} C_VEL
LIN {X 0,Y 509.326,Z 543.553,A -85,B 0,C 180,E1 -5497.134,E2 -5497.134} C_VEL
LIN {X 0,Y 509.497,Z 536.999,A -85,B 0,C 180,E1 -5498.527,E2 -5498.527} C_VEL
LIN {X 0,Y 509.714,Z 528.848,A -85,B 0,C 180,E1 -5499.924,E2 -5499.924} C_VEL
LIN {X 0,Y 509.966,Z 520.297,A -85,B 0,C 180,E1 -5501.124,E2 -5501.124} C_VEL
LIN {X 0,Y 510.321,Z 510.338,A -85,B 0,C 180,E1 -5502.285,E2 -5502.285} C_VEL
LIN {X 0,Y 510.663,Z 499.503,A -85,B 0,C 180,E1 -5503.328,E2 -5503.328} C_VEL
LIN {X 0,Y 511.048,Z 488.145,A -85,B 0,C 180,E1 -5504.23,E2 -5504.23} C_VEL
LIN {X 0,Y 511.472,Z 475.728,A -85,B 0,C 180,E1 -5505.032,E2 -5505.032} C_VEL
LIN {X 0,Y 511.879,Z 463.02,A -85,B 0,C 180,E1 -5505.682,E2 -5505.682} C_VEL
LIN {X 0,Y 512.141,Z 448.937,A -85,B 0,C 180,E1 -5506.23,E2 -5506.23} C_VEL
LIN {X 0,Y 512.445,Z 434.742,A -85,B 0,C 180,E1 -5506.611,E2 -5506.611} C_VEL
LIN {X 0,Y 512.624,Z 408.943,A -85,B 0,C 180,E1 -5507.015,E2 -5507.015} C_VEL
LIN {X 0,Y 513.246,Z 307.189,A -85,B 0,C 180,E1 -5508.496,E2 -5508.496} C_VEL
LIN {X 0,Y 511.417,Z 295.8,A -85,B 0,C 180,E1 -5508.752,E2 -5508.752} C_VEL
LIN {X 0,Y 512.297,Z 271.371,A -85,B 0,C 180,E1 -5511.952,E2 -5511.952} C_VEL
LIN {X 0,Y 512.812,Z 257.224,A -85,B 0,C 180,E1 -5513.846,E2 -5513.846} C_VEL
LIN {X 0,Y 509.921,Z 244.705,A -85,B 0,C 180,E1 -5515.772,E2 -5515.772} C_VEL
LIN {X 0,Y 509.876,Z 244.591,A -85,B 0,C 180,E1 -5518.844,E2 -5518.844} C_VEL
LIN {X 0,Y 509.82,Z 244.596,A -85,B 0,C 180,E1 -5521.59,E2 -5521.59} C_VEL
LIN {X 0,Y 509.845,Z 244.604,A -85,B 0,C 180,E1 -5524.413,E2 -5524.413} C_VEL
LIN {X 0,Y 509.814,Z 244.596,A -85,B 0,C 180,E1 -5527.34,E2 -5527.34} C_VEL
LIN {X 0,Y 509.835,Z 244.602,A -85,B 0,C 180,E1 -5530.382,E2 -5530.382} C_VEL
LIN {X 0,Y 509.836,Z 244.599,A -85,B 0,C 180,E1 -5533.064,E2 -5533.064} C_VEL
LIN {X 0,Y 509.826,Z 244.601,A -85,B 0,C 180,E1 -5535.792,E2 -5535.792} C_VEL
LIN {X 0,Y 509.854,Z 244.595,A -85,B 0,C 180,E1 -5538.574,E2 -5538.574} C_VEL
LIN {X 0,Y 509.847,Z 244.601,A -85,B 0,C 180,E1 -5541.786,E2 -5541.786} C_VEL
LIN {X 0,Y 509.841,Z 244.597,A -85,B 0,C 180,E1 -5544.623,E2 -5544.623} C_VEL
LIN {X 0,Y 509.86,Z 244.597,A -85,B 0,C 180,E1 -5547.481,E2 -5547.481} C_VEL
LIN {X 0,Y 509.875,Z 244.59,A -85,B 0,C 180,E1 -5550.269,E2 -5550.269} C_VEL
LIN {X 0,Y 509.88,Z 244.593,A -85,B 0,C 180,E1 -5552.944,E2 -5552.944} C_VEL
LIN {X 0,Y 509.863,Z 244.597,A -85,B 0,C 180,E1 -5555.574,E2 -5555.574} C_VEL
LIN {X 0,Y 509.816,Z 244.604,A -85,B 0,C 180,E1 -5558.148,E2 -5558.148} C_VEL
LIN {X 0,Y 509.858,Z 244.595,A -85,B 0,C 180,E1 -5560.682,E2 -5560.682} C_VEL
LIN {X 0,Y 509.881,Z 244.593,A -85,B 0,C 180,E1 -5563.175,E2 -5563.175} C_VEL
LIN {X 0,Y 509.858,Z 244.601,A -85,B 0,C 180,E1 -5565.634,E2 -5565.634} C_VEL
LIN {X 0,Y 509.906,Z 244.587,A -85,B 0,C 180,E1 -5568.875,E2 -5568.875} C_VEL
LIN {X 0,Y 509.945,Z 244.584,A -85,B 0,C 180,E1 -5572.079,E2 -5572.079} C_VEL
LIN {X 0,Y 509.976,Z 244.581,A -85,B 0,C 180,E1 -5574.464,E2 -5574.464} C_VEL
LIN {X 0,Y 510.048,Z 244.576,A -85,B 0,C 180,E1 -5577.631,E2 -5577.631} C_VEL
LIN {X 0,Y 510.058,Z 244.571,A -85,B 0,C 180,E1 -5580.79,E2 -5580.79} C_VEL
LIN {X 0,Y 509.951,Z 244.584,A -85,B 0,C 180,E1 -5583.16,E2 -5583.16} C_VEL
LIN {X 0,Y 509.972,Z 244.579,A -85,B 0,C 180,E1 -5586.33,E2 -5586.33} C_VEL
LIN {X 0,Y 509.91,Z 244.589,A -85,B 0,C 180,E1 -5588.721,E2 -5588.721} C_VEL
LIN {X 0,Y 509.898,Z 244.59,A -85,B 0,C 180,E1 -5591.932,E2 -5591.932} C_VEL
LIN {X 0,Y 509.888,Z 244.597,A -85,B 0,C 180,E1 -5595.242,E2 -5595.242} C_VEL
LIN {X 0,Y 509.883,Z 244.593,A -85,B 0,C 180,E1 -5598.002,E2 -5598.002} C_VEL
LIN {X 0,Y 509.845,Z 244.6,A -85,B 0,C 180,E1 -5601.002,E2 -5601.002} C_VEL
LIN {X 0,Y 509.865,Z 244.594,A -85,B 0,C 180,E1 -5604.427,E2 -5604.427} C_VEL
LIN {X 0,Y 509.881,Z 244.598,A -85,B 0,C 180,E1 -5607.056,E2 -5607.056} C_VEL
LIN {X 0,Y 509.853,Z 244.592,A -85,B 0,C 180,E1 -5609.752,E2 -5609.752} C_VEL
LIN {X 0,Y 509.873,Z 244.6,A -85,B 0,C 180,E1 -5612.776,E2 -5612.776} C_VEL
LIN {X 0,Y 509.84,Z 244.596,A -85,B 0,C 180,E1 -5615.582,E2 -5615.582} C_VEL
LIN {X 0,Y 509.849,Z 244.599,A -85,B 0,C 180,E1 -5618.339,E2 -5618.339} C_VEL
LIN {X 0,Y 509.855,Z 244.598,A -85,B 0,C 180,E1 -5621.426,E2 -5621.426} C_VEL
LIN {X 0,Y 509.856,Z 244.598,A -85,B 0,C 180,E1 -5624.669,E2 -5624.669} C_VEL
LIN {X 0,Y 509.861,Z 244.594,A -85,B 0,C 180,E1 -5628.104,E2 -5628.104} C_VEL
LIN {X 0,Y 509.846,Z 244.595,A -85,B 0,C 180,E1 -5630.648,E2 -5630.648} C_VEL
LIN {X 0,Y 509.821,Z 244.602,A -85,B 0,C 180,E1 -5633.742,E2 -5633.742} C_VEL
LIN {X 0,Y 509.153,Z 244.69,A -85,B 0,C 180,E1 -5634.402,E2 -5634.402} C_VEL
LIN {X 0,Y 506.339,Z 245.038,A -85,B 0,C 180,E1 -5635.474,E2 -5635.474} C_VEL
LIN {X 0,Y 503.952,Z 245.335,A -85,B 0,C 180,E1 -5636.337,E2 -5636.337} C_VEL
LIN {X 0,Y 502.905,Z 245.465,A -85,B 0,C 180,E1 -5637.003,E2 -5637.003} C_VEL
LIN {X 0,Y 502.808,Z 245.476,A -85,B 0,C 180,E1 -5637.229,E2 -5637.229} C_VEL
LIN {X 0,Y 502.817,Z 245.476,A -85,B 0,C 180,E1 -5640.066,E2 -5640.066} C_VEL
LIN {X 0,Y 502.862,Z 245.677,A -85,B 0,C 180,E1 -5641.288,E2 -5641.288} C_VEL
LIN {X 0,Y 505.366,Z 257.162,A -85,B 0,C 180,E1 -5643.278,E2 -5643.278} C_VEL
LIN {X 0,Y 505.326,Z 264.661,A -85,B 0,C 180,E1 -5644.46,E2 -5644.46} C_VEL
LIN {X 0,Y 504.581,Z 284.269,A -85,B 0,C 180,E1 -5647.479,E2 -5647.479} C_VEL
LIN {X 0,Y 503.822,Z 308.072,A -85,B 0,C 180,E1 -5651.076,E2 -5651.076} C_VEL
LIN {X 0,Y 503.656,Z 314.733,A -85,B 0,C 180,E1 -5652.041,E2 -5652.041} C_VEL
LIN {X 0,Y 505.846,Z 328.344,A -85,B 0,C 180,E1 -5652.333,E2 -5652.333} C_VEL
LIN {X 0,Y 505.391,Z 425.254,A -85,B 0,C 180,E1 -5653.683,E2 -5653.683} C_VEL
LIN {X 0,Y 505.159,Z 437.511,A -85,B 0,C 180,E1 -5654,E2 -5654} C_VEL
LIN {X 0,Y 504.842,Z 450.557,A -85,B 0,C 180,E1 -5654.508,E2 -5654.508} C_VEL
LIN {X 0,Y 504.454,Z 462.894,A -85,B 0,C 180,E1 -5655.167,E2 -5655.167} C_VEL
LIN {X 0,Y 503.974,Z 473.187,A -85,B 0,C 180,E1 -5655.875,E2 -5655.875} C_VEL
LIN {X 0,Y 503.614,Z 483.803,A -85,B 0,C 180,E1 -5656.791,E2 -5656.791} C_VEL
LIN {X 0,Y 503.23,Z 492.656,A -85,B 0,C 180,E1 -5657.724,E2 -5657.724} C_VEL
LIN {X 0,Y 502.9,Z 501.909,A -85,B 0,C 180,E1 -5658.922,E2 -5658.922} C_VEL
LIN {X 0,Y 502.592,Z 509.419,A -85,B 0,C 180,E1 -5660.137,E2 -5660.137} C_VEL
LIN {X 0,Y 502.37,Z 516.352,A -85,B 0,C 180,E1 -5661.553,E2 -5661.553} C_VEL
LIN {X 0,Y 502.247,Z 520.963,A -85,B 0,C 180,E1 -5662.765,E2 -5662.765} C_VEL
LIN {X 0,Y 502.164,Z 524.049,A -85,B 0,C 180,E1 -5663.804,E2 -5663.804} C_VEL
LIN {X 0,Y 502.066,Z 527.038,A -85,B 0,C 180,E1 -5665.182,E2 -5665.182} C_VEL
LIN {X 0,Y 502.128,Z 528.237,A -85,B 0,C 180,E1 -5665.987,E2 -5665.987} C_VEL
LIN {X 0,Y 502.112,Z 529.036,A -85,B 0,C 180,E1 -5666.79,E2 -5666.79} C_VEL
LIN {X 0,Y 502.037,Z 529.446,A -85,B 0,C 180,E1 -5668.396,E2 -5668.396} C_VEL
LIN {X 0,Y 501.987,Z 528.37,A -85,B 0,C 180,E1 -5670,E2 -5670} C_VEL
LIN {X 0,Y 502.064,Z 525.673,A -85,B 0,C 180,E1 -5671.604,E2 -5671.604} C_VEL
LIN {X 0,Y 502.214,Z 522.581,A -85,B 0,C 180,E1 -5672.807,E2 -5672.807} C_VEL
LIN {X 0,Y 502.305,Z 518.472,A -85,B 0,C 180,E1 -5674.011,E2 -5674.011} C_VEL
LIN {X 0,Y 502.534,Z 513.223,A -85,B 0,C 180,E1 -5675.215,E2 -5675.215} C_VEL
LIN {X 0,Y 502.685,Z 506.681,A -85,B 0,C 180,E1 -5676.422,E2 -5676.422} C_VEL
LIN {X 0,Y 502.999,Z 498.585,A -85,B 0,C 180,E1 -5677.628,E2 -5677.628} C_VEL
LIN {X 0,Y 503.399,Z 490.299,A -85,B 0,C 180,E1 -5678.631,E2 -5678.631} C_VEL
LIN {X 0,Y 503.782,Z 480.107,A -85,B 0,C 180,E1 -5679.637,E2 -5679.637} C_VEL
LIN {X 0,Y 504.104,Z 470.058,A -85,B 0,C 180,E1 -5680.442,E2 -5680.442} C_VEL
LIN {X 0,Y 504.532,Z 459.079,A -85,B 0,C 180,E1 -5681.144,E2 -5681.144} C_VEL
LIN {X 0,Y 504.925,Z 446.87,A -85,B 0,C 180,E1 -5681.745,E2 -5681.745} C_VEL
LIN {X 0,Y 505.216,Z 434.802,A -85,B 0,C 180,E1 -5682.171,E2 -5682.171} C_VEL
LIN {X 0,Y 505.389,Z 422.915,A -85,B 0,C 180,E1 -5682.447,E2 -5682.447} C_VEL
LIN {X 0,Y 505.686,Z 327.205,A -85,B 0,C 180,E1 -5683.776,E2 -5683.776} C_VEL
LIN {X 0,Y 503.665,Z 314.969,A -85,B 0,C 180,E1 -5684.031,E2 -5684.031} C_VEL
LIN {X 0,Y 503.696,Z 311.17,A -85,B 0,C 180,E1 -5684.545,E2 -5684.545} C_VEL
LIN {X 0,Y 504.382,Z 289.177,A -85,B 0,C 180,E1 -5687.851,E2 -5687.851} C_VEL
LIN {X 0,Y 505.118,Z 268.023,A -85,B 0,C 180,E1 -5691.079,E2 -5691.079} C_VEL
LIN {X 0,Y 505.41,Z 257.577,A -85,B 0,C 180,E1 -5692.698,E2 -5692.698} C_VEL
LIN {X 0,Y 502.82,Z 245.582,A -85,B 0,C 180,E1 -5694.753,E2 -5694.753} C_VEL
LIN {X 0,Y 502.834,Z 245.47,A -85,B 0,C 180,E1 -5697.466,E2 -5697.466} C_VEL
LIN {X 0,Y 502.812,Z 245.472,A -85,B 0,C 180,E1 -5700.21,E2 -5700.21} C_VEL
LIN {X 0,Y 502.833,Z 245.469,A -85,B 0,C 180,E1 -5703.03,E2 -5703.03} C_VEL
LIN {X 0,Y 502.774,Z 245.481,A -85,B 0,C 180,E1 -5705.95,E2 -5705.95} C_VEL
LIN {X 0,Y 502.801,Z 245.478,A -85,B 0,C 180,E1 -5708.975,E2 -5708.975} C_VEL
LIN {X 0,Y 502.83,Z 245.471,A -85,B 0,C 180,E1 -5712.135,E2 -5712.135} C_VEL
LIN {X 0,Y 502.799,Z 245.477,A -85,B 0,C 180,E1 -5715.467,E2 -5715.467} C_VEL
LIN {X 0,Y 502.818,Z 245.478,A -85,B 0,C 180,E1 -5718.933,E2 -5718.933} C_VEL
LIN {X 0,Y 502.792,Z 245.475,A -85,B 0,C 180,E1 -5722.045,E2 -5722.045} C_VEL
LIN {X 0,Y 502.806,Z 245.474,A -85,B 0,C 180,E1 -5725.034,E2 -5725.034} C_VEL
LIN {X 0,Y 502.784,Z 245.474,A -85,B 0,C 180,E1 -5727.915,E2 -5727.915} C_VEL
LIN {X 0,Y 502.833,Z 245.476,A -85,B 0,C 180,E1 -5730.712,E2 -5730.712} C_VEL
LIN {X 0,Y 502.858,Z 245.47,A -85,B 0,C 180,E1 -5733.438,E2 -5733.438} C_VEL
LIN {X 0,Y 502.786,Z 245.473,A -85,B 0,C 180,E1 -5736.086,E2 -5736.086} C_VEL
LIN {X 0,Y 502.778,Z 245.484,A -85,B 0,C 180,E1 -5738.688,E2 -5738.688} C_VEL
LIN {X 0,Y 502.825,Z 245.474,A -85,B 0,C 180,E1 -5741.248,E2 -5741.248} C_VEL
LIN {X 0,Y 502.817,Z 245.472,A -85,B 0,C 180,E1 -5743.767,E2 -5743.767} C_VEL
LIN {X 0,Y 502.829,Z 245.471,A -85,B 0,C 180,E1 -5746.254,E2 -5746.254} C_VEL
LIN {X 0,Y 502.87,Z 245.471,A -85,B 0,C 180,E1 -5748.716,E2 -5748.716} C_VEL
LIN {X 0,Y 502.895,Z 245.463,A -85,B 0,C 180,E1 -5751.966,E2 -5751.966} C_VEL
LIN {X 0,Y 502.932,Z 245.464,A -85,B 0,C 180,E1 -5754.386,E2 -5754.386} C_VEL
LIN {X 0,Y 503.018,Z 245.447,A -85,B 0,C 180,E1 -5757.597,E2 -5757.597} C_VEL
LIN {X 0,Y 503.019,Z 245.448,A -85,B 0,C 180,E1 -5760,E2 -5760} C_VEL
LIN {X 0,Y 503.017,Z 245.453,A -85,B 0,C 180,E1 -5762.402,E2 -5762.402} C_VEL
LIN {X 0,Y 502.931,Z 245.456,A -85,B 0,C 180,E1 -5765.613,E2 -5765.613} C_VEL
LIN {X 0,Y 502.894,Z 245.466,A -85,B 0,C 180,E1 -5768.033,E2 -5768.033} C_VEL
LIN {X 0,Y 502.869,Z 245.462,A -85,B 0,C 180,E1 -5771.283,E2 -5771.283} C_VEL
LIN {X 0,Y 502.838,Z 245.472,A -85,B 0,C 180,E1 -5774.571,E2 -5774.571} C_VEL
LIN {X 0,Y 502.855,Z 245.472,A -85,B 0,C 180,E1 -5777.907,E2 -5777.907} C_VEL
LIN {X 0,Y 502.821,Z 245.473,A -85,B 0,C 180,E1 -5780.536,E2 -5780.536} C_VEL
LIN {X 0,Y 502.79,Z 245.476,A -85,B 0,C 180,E1 -5783.04,E2 -5783.04} C_VEL
LIN {X 0,Y 502.833,Z 245.472,A -85,B 0,C 180,E1 -5785.676,E2 -5785.676} C_VEL
LIN {X 0,Y 502.836,Z 245.469,A -85,B 0,C 180,E1 -5788.373,E2 -5788.373} C_VEL
LIN {X 0,Y 502.791,Z 245.47,A -85,B 0,C 180,E1 -5791.5,E2 -5791.5} C_VEL
LIN {X 0,Y 502.8,Z 245.476,A -85,B 0,C 180,E1 -5794.445,E2 -5794.445} C_VEL
LIN {X 0,Y 502.776,Z 245.47,A -85,B 0,C 180,E1 -5797.179,E2 -5797.179} C_VEL
LIN {X 0,Y 502.783,Z 245.482,A -85,B 0,C 180,E1 -5800.016,E2 -5800.016} C_VEL
LIN {X 0,Y 502.798,Z 245.475,A -85,B 0,C 180,E1 -5802.2,E2 -5802.2} C_VEL
LIN {X 0,Y 502.797,Z 245.481,A -85,B 0,C 180,E1 -5805.469,E2 -5805.469} C_VEL
LIN {X 0,Y 502.816,Z 245.459,A -85,B 0,C 180,E1 -5808.935,E2 -5808.935} C_VEL
LIN {X 0,Y 502.79,Z 245.478,A -85,B 0,C 180,E1 -5812.047,E2 -5812.047} C_VEL
LIN {X 0,Y 502.796,Z 245.469,A -85,B 0,C 180,E1 -5815.035,E2 -5815.035} C_VEL
LIN {X 0,Y 502.783,Z 245.471,A -85,B 0,C 180,E1 -5817.916,E2 -5817.916} C_VEL
LIN {X 0,Y 502.823,Z 245.475,A -85,B 0,C 180,E1 -5820.713,E2 -5820.713} C_VEL
LIN {X 0,Y 502.885,Z 245.601,A -85,B 0,C 180,E1 -5824.022,E2 -5824.022} C_VEL
LIN {X 0,Y 505.882,Z 258.654,A -85,B 0,C 180,E1 -5826.024,E2 -5826.024} C_VEL
LIN {X 0,Y 505.402,Z 272.87,A -85,B 0,C 180,E1 -5827.948,E2 -5827.948} C_VEL
LIN {X 0,Y 504.54,Z 295.93,A -85,B 0,C 180,E1 -5831.008,E2 -5831.008} C_VEL
LIN {X 0,Y 506.585,Z 310.167,A -85,B 0,C 180,E1 -5831.319,E2 -5831.319} C_VEL
LIN {X 0,Y 505.598,Z 433.43,A -85,B 0,C 180,E1 -5833.158,E2 -5833.158} C_VEL
LIN {X 0,Y 505.342,Z 447.808,A -85,B 0,C 180,E1 -5833.54,E2 -5833.54} C_VEL
LIN {X 0,Y 504.989,Z 461.134,A -85,B 0,C 180,E1 -5834.048,E2 -5834.048} C_VEL
LIN {X 0,Y 504.531,Z 475.065,A -85,B 0,C 180,E1 -5834.757,E2 -5834.757} C_VEL
LIN {X 0,Y 504.098,Z 487.577,A -85,B 0,C 180,E1 -5835.57,E2 -5835.57} C_VEL
LIN {X 0,Y 503.666,Z 499.011,A -85,B 0,C 180,E1 -5836.484,E2 -5836.484} C_VEL
LIN {X 0,Y 503.275,Z 510.573,A -85,B 0,C 180,E1 -5837.613,E2 -5837.613} C_VEL
LIN {X 0,Y 502.929,Z 519.937,A -85,B 0,C 180,E1 -5838.718,E2 -5838.718} C_VEL
LIN {X 0,Y 502.666,Z 528.533,A -85,B 0,C 180,E1 -5839.935,E2 -5839.935} C_VEL
LIN {X 0,Y 502.417,Z 536.718,A -85,B 0,C 180,E1 -5841.352,E2 -5841.352} C_VEL
LIN {X 0,Y 502.252,Z 543.302,A -85,B 0,C 180,E1 -5842.765,E2 -5842.765} C_VEL
LIN {X 0,Y 502.171,Z 547.859,A -85,B 0,C 180,E1 -5843.975,E2 -5843.975} C_VEL
LIN {X 0,Y 502.102,Z 551.425,A -85,B 0,C 180,E1 -5845.183,E2 -5845.183} C_VEL
LIN {X 0,Y 502.112,Z 554.905,A -85,B 0,C 180,E1 -5846.791,E2 -5846.791} C_VEL
LIN {X 0,Y 502.033,Z 556.962,A -85,B 0,C 180,E1 -5848.396,E2 -5848.396} C_VEL
LIN {X 0,Y 501.979,Z 557.644,A -85,B 0,C 180,E1 -5850,E2 -5850} C_VEL
LIN {X 0,Y 502.033,Z 556.962,A -85,B 0,C 180,E1 -5851.604,E2 -5851.604} C_VEL
LIN {X 0,Y 502.112,Z 554.907,A -85,B 0,C 180,E1 -5853.21,E2 -5853.21} C_VEL
LIN {X 0,Y 502.102,Z 551.425,A -85,B 0,C 180,E1 -5854.817,E2 -5854.817} C_VEL
LIN {X 0,Y 502.234,Z 546.418,A -85,B 0,C 180,E1 -5856.428,E2 -5856.428} C_VEL
LIN {X 0,Y 502.352,Z 539.728,A -85,B 0,C 180,E1 -5858.042,E2 -5858.042} C_VEL
LIN {X 0,Y 502.535,Z 532.26,A -85,B 0,C 180,E1 -5859.458,E2 -5859.458} C_VEL
LIN {X 0,Y 502.794,Z 524.418,A -85,B 0,C 180,E1 -5860.673,E2 -5860.673} C_VEL
LIN {X 0,Y 503.138,Z 514.503,A -85,B 0,C 180,E1 -5861.944,E2 -5861.944} C_VEL
LIN {X 0,Y 503.427,Z 504.481,A -85,B 0,C 180,E1 -5863.009,E2 -5863.009} C_VEL
LIN {X 0,Y 503.901,Z 492.896,A -85,B 0,C 180,E1 -5864.024,E2 -5864.024} C_VEL
LIN {X 0,Y 504.397,Z 480.039,A -85,B 0,C 180,E1 -5864.937,E2 -5864.937} C_VEL
LIN {X 0,Y 504.822,Z 466.493,A -85,B 0,C 180,E1 -5865.7,E2 -5865.7} C_VEL
LIN {X 0,Y 505.179,Z 453.116,A -85,B 0,C 180,E1 -5866.276,E2 -5866.276} C_VEL
LIN {X 0,Y 505.485,Z 438.844,A -85,B 0,C 180,E1 -5866.718,E2 -5866.718} C_VEL
LIN {X 0,Y 505.708,Z 424.463,A -85,B 0,C 180,E1 -5866.994,E2 -5866.994} C_VEL
LIN {X 0,Y 506.566,Z 309.079,A -85,B 0,C 180,E1 -5868.699,E2 -5868.699} C_VEL
LIN {X 0,Y 504.539,Z 296.009,A -85,B 0,C 180,E1 -5868.992,E2 -5868.992} C_VEL
LIN {X 0,Y 505.479,Z 271.421,A -85,B 0,C 180,E1 -5872.264,E2 -5872.264} C_VEL
LIN {X 0,Y 505.958,Z 258.866,A -85,B 0,C 180,E1 -5873.972,E2 -5873.972} C_VEL
LIN {X 0,Y 502.888,Z 245.609,A -85,B 0,C 180,E1 -5876.034,E2 -5876.034} C_VEL
LIN {X 0,Y 502.823,Z 245.473,A -85,B 0,C 180,E1 -5879.287,E2 -5879.287} C_VEL
LIN {X 0,Y 502.783,Z 245.47,A -85,B 0,C 180,E1 -5882.084,E2 -5882.084} C_VEL
LIN {X 0,Y 502.797,Z 245.474,A -85,B 0,C 180,E1 -5884.965,E2 -5884.965} C_VEL
LIN {X 0,Y 502.79,Z 245.473,A -85,B 0,C 180,E1 -5887.953,E2 -5887.953} C_VEL
LIN {X 0,Y 502.817,Z 245.472,A -85,B 0,C 180,E1 -5891.065,E2 -5891.065} C_VEL
LIN {X 0,Y 502.778,Z 245.478,A -85,B 0,C 180,E1 -5893.375,E2 -5893.375} C_VEL
LIN {X 0,Y 502.786,Z 245.476,A -85,B 0,C 180,E1 -5895.661,E2 -5895.661} C_VEL
LIN {X 0,Y 502.815,Z 245.468,A -85,B 0,C 180,E1 -5899.005,E2 -5899.005} C_VEL
LIN {X 0,Y 502.789,Z 245.483,A -85,B 0,C 180,E1 -5902.046,E2 -5902.046} C_VEL
LIN {X 0,Y 502.805,Z 245.471,A -85,B 0,C 180,E1 -5905.035,E2 -5905.035} C_VEL
LIN {X 0,Y 502.783,Z 245.484,A -85,B 0,C 180,E1 -5907.915,E2 -5907.915} C_VEL
LIN {X 0,Y 502.831,Z 245.465,A -85,B 0,C 180,E1 -5910.713,E2 -5910.713} C_VEL
LIN {X 0,Y 502.856,Z 245.47,A -85,B 0,C 180,E1 -5913.439,E2 -5913.439} C_VEL
LIN {X 0,Y 502.786,Z 245.483,A -85,B 0,C 180,E1 -5916.086,E2 -5916.086} C_VEL
LIN {X 0,Y 502.777,Z 245.476,A -85,B 0,C 180,E1 -5918.689,E2 -5918.689} C_VEL
LIN {X 0,Y 502.824,Z 245.473,A -85,B 0,C 180,E1 -5921.248,E2 -5921.248} C_VEL
LIN {X 0,Y 502.817,Z 245.476,A -85,B 0,C 180,E1 -5923.767,E2 -5923.767} C_VEL
LIN {X 0,Y 502.825,Z 245.473,A -85,B 0,C 180,E1 -5926.255,E2 -5926.255} C_VEL
LIN {X 0,Y 502.87,Z 245.463,A -85,B 0,C 180,E1 -5928.717,E2 -5928.717} C_VEL
LIN {X 0,Y 502.895,Z 245.463,A -85,B 0,C 180,E1 -5931.967,E2 -5931.967} C_VEL
LIN {X 0,Y 502.932,Z 245.459,A -85,B 0,C 180,E1 -5934.387,E2 -5934.387} C_VEL
LIN {X 0,Y 503.018,Z 245.451,A -85,B 0,C 180,E1 -5937.598,E2 -5937.598} C_VEL
LIN {X 0,Y 503.02,Z 245.45,A -85,B 0,C 180,E1 -5940,E2 -5940} C_VEL
LIN {X 0,Y 503.018,Z 245.444,A -85,B 0,C 180,E1 -5942.403,E2 -5942.403} C_VEL
LIN {X 0,Y 502.932,Z 245.462,A -85,B 0,C 180,E1 -5945.614,E2 -5945.614} C_VEL
LIN {X 0,Y 502.895,Z 245.463,A -85,B 0,C 180,E1 -5948.034,E2 -5948.034} C_VEL
LIN {X 0,Y 502.871,Z 245.47,A -85,B 0,C 180,E1 -5951.284,E2 -5951.284} C_VEL
LIN {X 0,Y 502.839,Z 245.47,A -85,B 0,C 180,E1 -5954.571,E2 -5954.571} C_VEL
LIN {X 0,Y 502.857,Z 245.469,A -85,B 0,C 180,E1 -5957.908,E2 -5957.908} C_VEL
LIN {X 0,Y 502.823,Z 245.47,A -85,B 0,C 180,E1 -5960.537,E2 -5960.537} C_VEL
LIN {X 0,Y 502.789,Z 245.483,A -85,B 0,C 180,E1 -5963.041,E2 -5963.041} C_VEL
LIN {X 0,Y 502.836,Z 245.473,A -85,B 0,C 180,E1 -5965.676,E2 -5965.676} C_VEL
LIN {X 0,Y 502.836,Z 245.465,A -85,B 0,C 180,E1 -5968.373,E2 -5968.373} C_VEL
LIN {X 0,Y 502.793,Z 245.479,A -85,B 0,C 180,E1 -5971.5,E2 -5971.5} C_VEL
LIN {X 0,Y 502.803,Z 245.473,A -85,B 0,C 180,E1 -5974.445,E2 -5974.445} C_VEL
LIN {X 0,Y 502.779,Z 245.483,A -85,B 0,C 180,E1 -5977.179,E2 -5977.179} C_VEL
LIN {X 0,Y 502.786,Z 245.47,A -85,B 0,C 180,E1 -5980.016,E2 -5980.016} C_VEL
LIN {X 0,Y 502.801,Z 245.476,A -85,B 0,C 180,E1 -5982.2,E2 -5982.2} C_VEL
LIN {X 0,Y 502.8,Z 245.477,A -85,B 0,C 180,E1 -5985.469,E2 -5985.469} C_VEL
LIN {X 0,Y 502.83,Z 245.468,A -85,B 0,C 180,E1 -5987.865,E2 -5987.865} C_VEL
LIN {X 0,Y 502.802,Z 245.466,A -85,B 0,C 180,E1 -5991.025,E2 -5991.025} C_VEL
LIN {X 0,Y 502.776,Z 245.482,A -85,B 0,C 180,E1 -5994.17,E2 -5994.17} C_VEL
LIN {X 0,Y 502.808,Z 245.476,A -85,B 0,C 180,E1 -5997.229,E2 -5997.229} C_VEL
LIN {X 0,Y 502.109,Z 245.571,A -85,B 0,C 180,E1 -5997.898,E2 -5997.898} C_VEL
LIN {X 0,Y 499.253,Z 245.913,A -85,B 0,C 180,E1 -5998.984,E2 -5998.984} C_VEL
LIN {X 0,Y 496.868,Z 246.214,A -85,B 0,C 180,E1 -5999.859,E2 -5999.859} C_VEL
LIN {X 0,Y 495.858,Z 246.346,A -85,B 0,C 180,E1 -6000.534,E2 -6000.534} C_VEL
LIN {X 0,Y 495.782,Z 246.364,A -85,B 0,C 180,E1 -6000.763,E2 -6000.763} C_VEL
LIN {X 0,Y 495.823,Z 246.551,A -85,B 0,C 180,E1 -6001.015,E2 -6001.015} C_VEL
LIN {X 0,Y 498.523,Z 258.869,A -85,B 0,C 180,E1 -6003.185,E2 -6003.185} C_VEL
LIN {X 0,Y 498.452,Z 266.186,A -85,B 0,C 180,E1 -6004.353,E2 -6004.353} C_VEL
LIN {X 0,Y 497.61,Z 286.903,A -85,B 0,C 180,E1 -6007.584,E2 -6007.584} C_VEL
LIN {X 0,Y 496.847,Z 309.322,A -85,B 0,C 180,E1 -6011.014,E2 -6011.014} C_VEL
LIN {X 0,Y 496.72,Z 314.622,A -85,B 0,C 180,E1 -6011.786,E2 -6011.786} C_VEL
LIN {X 0,Y 499.088,Z 329.231,A -85,B 0,C 180,E1 -6012.1,E2 -6012.1} C_VEL
LIN {X 0,Y 498.584,Z 425.746,A -85,B 0,C 180,E1 -6013.46,E2 -6013.46} C_VEL
LIN {X 0,Y 498.338,Z 438.391,A -85,B 0,C 180,E1 -6013.798,E2 -6013.798} C_VEL
LIN {X 0,Y 498.02,Z 450.884,A -85,B 0,C 180,E1 -6014.295,E2 -6014.295} C_VEL
LIN {X 0,Y 497.581,Z 463.098,A -85,B 0,C 180,E1 -6014.958,E2 -6014.958} C_VEL
LIN {X 0,Y 497.047,Z 474.665,A -85,B 0,C 180,E1 -6015.779,E2 -6015.779} C_VEL
LIN {X 0,Y 496.643,Z 485.049,A -85,B 0,C 180,E1 -6016.706,E2 -6016.706} C_VEL
LIN {X 0,Y 496.153,Z 494.893,A -85,B 0,C 180,E1 -6017.794,E2 -6017.794} C_VEL
LIN {X 0,Y 495.86,Z 503.418,A -85,B 0,C 180,E1 -6018.969,E2 -6018.969} C_VEL
LIN {X 0,Y 495.518,Z 510.68,A -85,B 0,C 180,E1 -6020.201,E2 -6020.201} C_VEL
LIN {X 0,Y 495.326,Z 516.508,A -85,B 0,C 180,E1 -6021.432,E2 -6021.432} C_VEL
LIN {X 0,Y 495.171,Z 521.119,A -85,B 0,C 180,E1 -6022.661,E2 -6022.661} C_VEL
LIN {X 0,Y 495.125,Z 523.716,A -85,B 0,C 180,E1 -6023.523,E2 -6023.523} C_VEL
LIN {X 0,Y 494.991,Z 527.204,A -85,B 0,C 180,E1 -6025.113,E2 -6025.113} C_VEL
LIN {X 0,Y 495.025,Z 528.408,A -85,B 0,C 180,E1 -6025.929,E2 -6025.929} C_VEL
LIN {X 0,Y 495.034,Z 529.22,A -85,B 0,C 180,E1 -6026.745,E2 -6026.745} C_VEL
LIN {X 0,Y 494.963,Z 529.649,A -85,B 0,C 180,E1 -6028.373,E2 -6028.373} C_VEL
LIN {X 0,Y 494.905,Z 528.606,A -85,B 0,C 180,E1 -6030,E2 -6030} C_VEL
LIN {X 0,Y 494.99,Z 525.954,A -85,B 0,C 180,E1 -6031.627,E2 -6031.627} C_VEL
LIN {X 0,Y 495.152,Z 522.903,A -85,B 0,C 180,E1 -6032.847,E2 -6032.847} C_VEL
LIN {X 0,Y 495.248,Z 518.844,A -85,B 0,C 180,E1 -6034.069,E2 -6034.069} C_VEL
LIN {X 0,Y 495.481,Z 513.653,A -85,B 0,C 180,E1 -6035.29,E2 -6035.29} C_VEL
LIN {X 0,Y 495.661,Z 507.178,A -85,B 0,C 180,E1 -6036.513,E2 -6036.513} C_VEL
LIN {X 0,Y 495.986,Z 499.157,A -85,B 0,C 180,E1 -6037.736,E2 -6037.736} C_VEL
LIN {X 0,Y 496.436,Z 490.961,A -85,B 0,C 180,E1 -6038.753,E2 -6038.753} C_VEL
LIN {X 0,Y 496.847,Z 480.922,A -85,B 0,C 180,E1 -6039.773,E2 -6039.773} C_VEL
LIN {X 0,Y 497.28,Z 469.603,A -85,B 0,C 180,E1 -6040.69,E2 -6040.69} C_VEL
LIN {X 0,Y 497.716,Z 458.461,A -85,B 0,C 180,E1 -6041.401,E2 -6041.401} C_VEL
LIN {X 0,Y 498.131,Z 445.883,A -85,B 0,C 180,E1 -6042.011,E2 -6042.011} C_VEL
LIN {X 0,Y 498.418,Z 433.259,A -85,B 0,C 180,E1 -6042.443,E2 -6042.443} C_VEL
LIN {X 0,Y 498.619,Z 420.168,A -85,B 0,C 180,E1 -6042.722,E2 -6042.722} C_VEL
LIN {X 0,Y 498.947,Z 328.398,A -85,B 0,C 180,E1 -6043.994,E2 -6043.994} C_VEL
LIN {X 0,Y 496.717,Z 314.713,A -85,B 0,C 180,E1 -6044.283,E2 -6044.283} C_VEL
LIN {X 0,Y 497.104,Z 298.95,A -85,B 0,C 180,E1 -6046.636,E2 -6046.636} C_VEL
LIN {X 0,Y 497.83,Z 279.692,A -85,B 0,C 180,E1 -6049.589,E2 -6049.589} C_VEL
LIN {X 0,Y 498.628,Z 260.437,A -85,B 0,C 180,E1 -6052.586,E2 -6052.586} C_VEL
LIN {X 0,Y 497.099,Z 252.343,A -85,B 0,C 180,E1 -6053.961,E2 -6053.961} C_VEL
LIN {X 0,Y 495.768,Z 246.435,A -85,B 0,C 180,E1 -6055.021,E2 -6055.021} C_VEL
LIN {X 0,Y 495.816,Z 246.337,A -85,B 0,C 180,E1 -6056.974,E2 -6056.974} C_VEL
LIN {X 0,Y 495.767,Z 246.349,A -85,B 0,C 180,E1 -6060.146,E2 -6060.146} C_VEL
LIN {X 0,Y 495.794,Z 246.343,A -85,B 0,C 180,E1 -6063.244,E2 -6063.244} C_VEL
LIN {X 0,Y 495.72,Z 246.36,A -85,B 0,C 180,E1 -6066.088,E2 -6066.088} C_VEL
LIN {X 0,Y 495.763,Z 246.353,A -85,B 0,C 180,E1 -6068.767,E2 -6068.767} C_VEL
LIN {X 0,Y 495.777,Z 246.352,A -85,B 0,C 180,E1 -6071.778,E2 -6071.778} C_VEL
LIN {X 0,Y 495.748,Z 246.354,A -85,B 0,C 180,E1 -6075.138,E2 -6075.138} C_VEL
LIN {X 0,Y 495.754,Z 246.352,A -85,B 0,C 180,E1 -6078.218,E2 -6078.218} C_VEL
LIN {X 0,Y 495.749,Z 246.357,A -85,B 0,C 180,E1 -6081.408,E2 -6081.408} C_VEL
LIN {X 0,Y 495.754,Z 246.353,A -85,B 0,C 180,E1 -6084.462,E2 -6084.462} C_VEL
LIN {X 0,Y 495.766,Z 246.351,A -85,B 0,C 180,E1 -6087.405,E2 -6087.405} C_VEL
LIN {X 0,Y 495.777,Z 246.351,A -85,B 0,C 180,E1 -6090.254,E2 -6090.254} C_VEL
LIN {X 0,Y 495.819,Z 246.349,A -85,B 0,C 180,E1 -6093.25,E2 -6093.25} C_VEL
LIN {X 0,Y 495.747,Z 246.35,A -85,B 0,C 180,E1 -6095.724,E2 -6095.724} C_VEL
LIN {X 0,Y 495.737,Z 246.357,A -85,B 0,C 180,E1 -6098.37,E2 -6098.37} C_VEL
LIN {X 0,Y 495.779,Z 246.355,A -85,B 0,C 180,E1 -6100.971,E2 -6100.971} C_VEL
LIN {X 0,Y 495.775,Z 246.349,A -85,B 0,C 180,E1 -6103.529,E2 -6103.529} C_VEL
LIN {X 0,Y 495.79,Z 246.346,A -85,B 0,C 180,E1 -6106.055,E2 -6106.055} C_VEL
LIN {X 0,Y 495.845,Z 246.349,A -85,B 0,C 180,E1 -6108.554,E2 -6108.554} C_VEL
LIN {X 0,Y 495.866,Z 246.338,A -85,B 0,C 180,E1 -6111.852,E2 -6111.852} C_VEL
LIN {X 0,Y 495.889,Z 246.34,A -85,B 0,C 180,E1 -6114.306,E2 -6114.306} C_VEL
LIN {X 0,Y 495.987,Z 246.323,A -85,B 0,C 180,E1 -6117.563,E2 -6117.563} C_VEL
LIN {X 0,Y 495.991,Z 246.324,A -85,B 0,C 180,E1 -6120,E2 -6120} C_VEL
LIN {X 0,Y 495.986,Z 246.33,A -85,B 0,C 180,E1 -6122.436,E2 -6122.436} C_VEL
LIN {X 0,Y 495.889,Z 246.333,A -85,B 0,C 180,E1 -6125.693,E2 -6125.693} C_VEL
LIN {X 0,Y 495.866,Z 246.343,A -85,B 0,C 180,E1 -6128.148,E2 -6128.148} C_VEL
LIN {X 0,Y 495.844,Z 246.337,A -85,B 0,C 180,E1 -6131.445,E2 -6131.445} C_VEL
LIN {X 0,Y 495.783,Z 246.348,A -85,B 0,C 180,E1 -6134.783,E2 -6134.783} C_VEL
LIN {X 0,Y 495.781,Z 246.348,A -85,B 0,C 180,E1 -6137.319,E2 -6137.319} C_VEL
LIN {X 0,Y 495.765,Z 246.356,A -85,B 0,C 180,E1 -6139.89,E2 -6139.89} C_VEL
LIN {X 0,Y 495.758,Z 246.352,A -85,B 0,C 180,E1 -6142.863,E2 -6142.863} C_VEL
LIN {X 0,Y 495.785,Z 246.356,A -85,B 0,C 180,E1 -6146.068,E2 -6146.068} C_VEL
LIN {X 0,Y 495.774,Z 246.346,A -85,B 0,C 180,E1 -6148.815,E2 -6148.815} C_VEL
LIN {X 0,Y 495.753,Z 246.349,A -85,B 0,C 180,E1 -6151.726,E2 -6151.726} C_VEL
LIN {X 0,Y 495.771,Z 246.35,A -85,B 0,C 180,E1 -6154.696,E2 -6154.696} C_VEL
LIN {X 0,Y 495.726,Z 246.352,A -85,B 0,C 180,E1 -6157.562,E2 -6157.562} C_VEL
LIN {X 0,Y 495.762,Z 246.351,A -85,B 0,C 180,E1 -6160.7,E2 -6160.7} C_VEL
LIN {X 0,Y 495.729,Z 246.361,A -85,B 0,C 180,E1 -6164.001,E2 -6164.001} C_VEL
LIN {X 0,Y 495.722,Z 246.35,A -85,B 0,C 180,E1 -6167.117,E2 -6167.117} C_VEL
LIN {X 0,Y 495.755,Z 246.353,A -85,B 0,C 180,E1 -6169.953,E2 -6169.953} C_VEL
LIN {X 0,Y 495.724,Z 246.355,A -85,B 0,C 180,E1 -6172.554,E2 -6172.554} C_VEL
LIN {X 0,Y 495.775,Z 246.349,A -85,B 0,C 180,E1 -6175.457,E2 -6175.457} C_VEL
LIN {X 0,Y 495.754,Z 246.344,A -85,B 0,C 180,E1 -6178.364,E2 -6178.364} C_VEL
LIN {X 0,Y 495.787,Z 246.346,A -85,B 0,C 180,E1 -6181.507,E2 -6181.507} C_VEL
LIN {X 0,Y 495.852,Z 246.484,A -85,B 0,C 180,E1 -6183.757,E2 -6183.757} C_VEL
LIN {X 0,Y 498.998,Z 260.189,A -85,B 0,C 180,E1 -6185.893,E2 -6185.893} C_VEL
LIN {X 0,Y 498.765,Z 269.664,A -85,B 0,C 180,E1 -6187.202,E2 -6187.202} C_VEL
LIN {X 0,Y 497.847,Z 288.564,A -85,B 0,C 180,E1 -6189.766,E2 -6189.766} C_VEL
LIN {X 0,Y 497.632,Z 296.069,A -85,B 0,C 180,E1 -6190.761,E2 -6190.761} C_VEL
LIN {X 0,Y 499.799,Z 309.844,A -85,B 0,C 180,E1 -6191.078,E2 -6191.078} C_VEL
LIN {X 0,Y 498.76,Z 433.099,A -85,B 0,C 180,E1 -6192.947,E2 -6192.947} C_VEL
LIN {X 0,Y 498.443,Z 447.465,A -85,B 0,C 180,E1 -6193.33,E2 -6193.33} C_VEL
LIN {X 0,Y 498.088,Z 461.458,A -85,B 0,C 180,E1 -6193.875,E2 -6193.875} C_VEL
LIN {X 0,Y 497.642,Z 474.37,A -85,B 0,C 180,E1 -6194.54,E2 -6194.54} C_VEL
LIN {X 0,Y 497.131,Z 486.98,A -85,B 0,C 180,E1 -6195.363,E2 -6195.363} C_VEL
LIN {X 0,Y 496.713,Z 498.497,A -85,B 0,C 180,E1 -6196.291,E2 -6196.291} C_VEL
LIN {X 0,Y 496.303,Z 509.064,A -85,B 0,C 180,E1 -6197.321,E2 -6197.321} C_VEL
LIN {X 0,Y 495.906,Z 519.553,A -85,B 0,C 180,E1 -6198.556,E2 -6198.556} C_VEL
LIN {X 0,Y 495.601,Z 528.191,A -85,B 0,C 180,E1 -6199.79,E2 -6199.79} C_VEL
LIN {X 0,Y 495.355,Z 536.417,A -85,B 0,C 180,E1 -6201.227,E2 -6201.227} C_VEL
LIN {X 0,Y 495.173,Z 543.031,A -85,B 0,C 180,E1 -6202.661,E2 -6202.661} C_VEL
LIN {X 0,Y 495.087,Z 547.288,A -85,B 0,C 180,E1 -6203.795,E2 -6203.795} C_VEL
LIN {X 0,Y 495.029,Z 551.193,A -85,B 0,C 180,E1 -6205.114,E2 -6205.114} C_VEL
LIN {X 0,Y 495.033,Z 554.691,A -85,B 0,C 180,E1 -6206.745,E2 -6206.745} C_VEL
LIN {X 0,Y 494.959,Z 556.759,A -85,B 0,C 180,E1 -6208.373,E2 -6208.373} C_VEL
LIN {X 0,Y 494.896,Z 557.446,A -85,B 0,C 180,E1 -6210,E2 -6210} C_VEL
LIN {X 0,Y 494.959,Z 556.76,A -85,B 0,C 180,E1 -6211.627,E2 -6211.627} C_VEL
LIN {X 0,Y 495.033,Z 554.693,A -85,B 0,C 180,E1 -6213.255,E2 -6213.255} C_VEL
LIN {X 0,Y 495.029,Z 551.195,A -85,B 0,C 180,E1 -6214.886,E2 -6214.886} C_VEL
LIN {X 0,Y 495.129,Z 546.284,A -85,B 0,C 180,E1 -6216.486,E2 -6216.486} C_VEL
LIN {X 0,Y 495.208,Z 541.283,A -85,B 0,C 180,E1 -6217.748,E2 -6217.748} C_VEL
LIN {X 0,Y 495.415,Z 534.219,A -85,B 0,C 180,E1 -6219.183,E2 -6219.183} C_VEL
LIN {X 0,Y 495.699,Z 525.436,A -85,B 0,C 180,E1 -6220.621,E2 -6220.621} C_VEL
LIN {X 0,Y 496.071,Z 515.839,A -85,B 0,C 180,E1 -6221.904,E2 -6221.904} C_VEL
LIN {X 0,Y 496.409,Z 505.064,A -85,B 0,C 180,E1 -6223.092,E2 -6223.092} C_VEL
LIN {X 0,Y 496.896,Z 493.645,A -85,B 0,C 180,E1 -6224.121,E2 -6224.121} C_VEL
LIN {X 0,Y 497.416,Z 480.998,A -85,B 0,C 180,E1 -6225.047,E2 -6225.047} C_VEL
LIN {X 0,Y 497.883,Z 467.174,A -85,B 0,C 180,E1 -6225.85,E2 -6225.85} C_VEL
LIN {X 0,Y 498.291,Z 453.756,A -85,B 0,C 180,E1 -6226.446,E2 -6226.446} C_VEL
LIN {X 0,Y 498.599,Z 439.771,A -85,B 0,C 180,E1 -6226.898,E2 -6226.898} C_VEL
LIN {X 0,Y 498.836,Z 426.146,A -85,B 0,C 180,E1 -6227.18,E2 -6227.18} C_VEL
LIN {X 0,Y 499.733,Z 308.984,A -85,B 0,C 180,E1 -6228.95,E2 -6228.95} C_VEL
LIN {X 0,Y 497.685,Z 296.138,A -85,B 0,C 180,E1 -6229.247,E2 -6229.247} C_VEL
LIN {X 0,Y 498.702,Z 271.481,A -85,B 0,C 180,E1 -6232.583,E2 -6232.583} C_VEL
LIN {X 0,Y 499.104,Z 260.513,A -85,B 0,C 180,E1 -6234.101,E2 -6234.101} C_VEL
LIN {X 0,Y 495.859,Z 246.486,A -85,B 0,C 180,E1 -6236.319,E2 -6236.319} C_VEL
LIN {X 0,Y 495.771,Z 246.346,A -85,B 0,C 180,E1 -6238.814,E2 -6238.814} C_VEL
LIN {X 0,Y 495.754,Z 246.345,A -85,B 0,C 180,E1 -6241.725,E2 -6241.725} C_VEL
LIN {X 0,Y 495.766,Z 246.352,A -85,B 0,C 180,E1 -6244.693,E2 -6244.693} C_VEL
LIN {X 0,Y 495.726,Z 246.35,A -85,B 0,C 180,E1 -6247.561,E2 -6247.561} C_VEL
LIN {X 0,Y 495.763,Z 246.353,A -85,B 0,C 180,E1 -6250.699,E2 -6250.699} C_VEL
LIN {X 0,Y 495.731,Z 246.357,A -85,B 0,C 180,E1 -6253.695,E2 -6253.695} C_VEL
LIN {X 0,Y 495.724,Z 246.364,A -85,B 0,C 180,E1 -6256.305,E2 -6256.305} C_VEL
LIN {X 0,Y 495.762,Z 246.346,A -85,B 0,C 180,E1 -6259.3,E2 -6259.3} C_VEL
LIN {X 0,Y 495.727,Z 246.356,A -85,B 0,C 180,E1 -6262.438,E2 -6262.438} C_VEL
LIN {X 0,Y 495.78,Z 246.347,A -85,B 0,C 180,E1 -6265.457,E2 -6265.457} C_VEL
LIN {X 0,Y 495.754,Z 246.352,A -85,B 0,C 180,E1 -6268.364,E2 -6268.364} C_VEL
LIN {X 0,Y 495.783,Z 246.344,A -85,B 0,C 180,E1 -6271.506,E2 -6271.506} C_VEL
LIN {X 0,Y 495.785,Z 246.357,A -85,B 0,C 180,E1 -6273.932,E2 -6273.932} C_VEL
LIN {X 0,Y 495.759,Z 246.352,A -85,B 0,C 180,E1 -6277.137,E2 -6277.137} C_VEL
LIN {X 0,Y 495.766,Z 246.356,A -85,B 0,C 180,E1 -6280.11,E2 -6280.11} C_VEL
LIN {X 0,Y 495.781,Z 246.348,A -85,B 0,C 180,E1 -6282.681,E2 -6282.681} C_VEL
LIN {X 0,Y 495.783,Z 246.349,A -85,B 0,C 180,E1 -6285.217,E2 -6285.217} C_VEL
LIN {X 0,Y 495.844,Z 246.339,A -85,B 0,C 180,E1 -6288.555,E2 -6288.555} C_VEL
LIN {X 0,Y 495.866,Z 246.34,A -85,B 0,C 180,E1 -6291.852,E2 -6291.852} C_VEL
LIN {X 0,Y 495.89,Z 246.336,A -85,B 0,C 180,E1 -6294.307,E2 -6294.307} C_VEL
LIN {X 0,Y 495.987,Z 246.327,A -85,B 0,C 180,E1 -6297.564,E2 -6297.564} C_VEL
LIN {X 0,Y 495.991,Z 246.325,A -85,B 0,C 180,E1 -6300,E2 -6300} C_VEL
LIN {X 0,Y 495.987,Z 246.319,A -85,B 0,C 180,E1 -6302.437,E2 -6302.437} C_VEL
LIN {X 0,Y 495.89,Z 246.338,A -85,B 0,C 180,E1 -6305.694,E2 -6305.694} C_VEL
LIN {X 0,Y 495.867,Z 246.338,A -85,B 0,C 180,E1 -6308.148,E2 -6308.148} C_VEL
LIN {X 0,Y 495.845,Z 246.344,A -85,B 0,C 180,E1 -6311.446,E2 -6311.446} C_VEL
LIN {X 0,Y 495.784,Z 246.35,A -85,B 0,C 180,E1 -6314.783,E2 -6314.783} C_VEL
LIN {X 0,Y 495.783,Z 246.356,A -85,B 0,C 180,E1 -6317.319,E2 -6317.319} C_VEL
LIN {X 0,Y 495.767,Z 246.349,A -85,B 0,C 180,E1 -6319.891,E2 -6319.891} C_VEL
LIN {X 0,Y 495.757,Z 246.357,A -85,B 0,C 180,E1 -6322.862,E2 -6322.862} C_VEL
LIN {X 0,Y 495.786,Z 246.349,A -85,B 0,C 180,E1 -6326.069,E2 -6326.069} C_VEL
LIN {X 0,Y 495.768,Z 246.347,A -85,B 0,C 180,E1 -6328.815,E2 -6328.815} C_VEL
LIN {X 0,Y 495.755,Z 246.354,A -85,B 0,C 180,E1 -6331.727,E2 -6331.727} C_VEL
LIN {X 0,Y 495.774,Z 246.349,A -85,B 0,C 180,E1 -6334.696,E2 -6334.696} C_VEL
LIN {X 0,Y 495.729,Z 246.357,A -85,B 0,C 180,E1 -6337.562,E2 -6337.562} C_VEL
LIN {X 0,Y 495.765,Z 246.35,A -85,B 0,C 180,E1 -6340.701,E2 -6340.701} C_VEL
LIN {X 0,Y 495.733,Z 246.352,A -85,B 0,C 180,E1 -6344.002,E2 -6344.002} C_VEL
LIN {X 0,Y 495.734,Z 246.355,A -85,B 0,C 180,E1 -6347.119,E2 -6347.119} C_VEL
LIN {X 0,Y 495.759,Z 246.353,A -85,B 0,C 180,E1 -6349.954,E2 -6349.954} C_VEL
LIN {X 0,Y 495.728,Z 246.347,A -85,B 0,C 180,E1 -6352.554,E2 -6352.554} C_VEL
LIN {X 0,Y 495.772,Z 246.345,A -85,B 0,C 180,E1 -6355.457,E2 -6355.457} C_VEL
LIN {X 0,Y 495.756,Z 246.354,A -85,B 0,C 180,E1 -6358.364,E2 -6358.364} C_VEL
LIN {X 0,Y 495.782,Z 246.364,A -85,B 0,C 180,E1 -6360.763,E2 -6360.763} C_VEL
LIN {X 0,Y 495.69,Z 247.236,A -85,B 0,C 180,E1 -6361.109,E2 -6361.109} C_VEL
LIN {X 0,Y 495.19,Z 250.345,A -85,B 0,C 180,E1 -6361.613,E2 -6361.613} C_VEL
LIN {X 0,Y 491.989,Z 262.314,A -85,B 0,C 180,E1 -6363.377,E2 -6363.377} C_VEL
LIN {X 0,Y 491.75,Z 264.568,A -85,B 0,C 180,E1 -6363.742,E2 -6363.742} C_VEL
LIN {X 0,Y 490.888,Z 283.948,A -85,B 0,C 180,E1 -6366.815,E2 -6366.815} C_VEL
LIN {X 0,Y 489.971,Z 306.37,A -85,B 0,C 180,E1 -6370.301,E2 -6370.301} C_VEL
LIN {X 0,Y 489.778,Z 314.478,A -85,B 0,C 180,E1 -6371.52,E2 -6371.52} C_VEL
LIN {X 0,Y 492.322,Z 329.964,A -85,B 0,C 180,E1 -6371.858,E2 -6371.858} C_VEL
LIN {X 0,Y 491.813,Z 424.858,A -85,B 0,C 180,E1 -6373.201,E2 -6373.201} C_VEL
LIN {X 0,Y 491.537,Z 437.804,A -85,B 0,C 180,E1 -6373.54,E2 -6373.54} C_VEL
LIN {X 0,Y 491.205,Z 451.205,A -85,B 0,C 180,E1 -6374.078,E2 -6374.078} C_VEL
LIN {X 0,Y 490.731,Z 463.272,A -85,B 0,C 180,E1 -6374.743,E2 -6374.743} C_VEL
LIN {X 0,Y 490.139,Z 474.839,A -85,B 0,C 180,E1 -6375.574,E2 -6375.574} C_VEL
LIN {X 0,Y 489.698,Z 485.221,A -85,B 0,C 180,E1 -6376.514,E2 -6376.514} C_VEL
LIN {X 0,Y 489.251,Z 494.579,A -85,B 0,C 180,E1 -6377.557,E2 -6377.557} C_VEL
LIN {X 0,Y 488.864,Z 503.585,A -85,B 0,C 180,E1 -6378.809,E2 -6378.809} C_VEL
LIN {X 0,Y 488.486,Z 510.842,A -85,B 0,C 180,E1 -6380.058,E2 -6380.058} C_VEL
LIN {X 0,Y 488.278,Z 516.667,A -85,B 0,C 180,E1 -6381.308,E2 -6381.308} C_VEL
LIN {X 0,Y 488.122,Z 521.275,A -85,B 0,C 180,E1 -6382.555,E2 -6382.555} C_VEL
LIN {X 0,Y 488.043,Z 524.14,A -85,B 0,C 180,E1 -6383.532,E2 -6383.532} C_VEL
LIN {X 0,Y 487.917,Z 527.37,A -85,B 0,C 180,E1 -6385.042,E2 -6385.042} C_VEL
LIN {X 0,Y 487.957,Z 529.402,A -85,B 0,C 180,E1 -6386.697,E2 -6386.697} C_VEL
LIN {X 0,Y 487.891,Z 529.853,A -85,B 0,C 180,E1 -6388.349,E2 -6388.349} C_VEL
LIN {X 0,Y 487.825,Z 528.837,A -85,B 0,C 180,E1 -6390,E2 -6390} C_VEL
LIN {X 0,Y 487.843,Z 527.743,A -85,B 0,C 180,E1 -6390.825,E2 -6390.825} C_VEL
LIN {X 0,Y 488.034,Z 524.333,A -85,B 0,C 180,E1 -6392.476,E2 -6392.476} C_VEL
LIN {X 0,Y 488.202,Z 520.658,A -85,B 0,C 180,E1 -6393.714,E2 -6393.714} C_VEL
LIN {X 0,Y 488.415,Z 515.908,A -85,B 0,C 180,E1 -6394.953,E2 -6394.953} C_VEL
LIN {X 0,Y 488.462,Z 509.957,A -85,B 0,C 180,E1 -6396.195,E2 -6396.195} C_VEL
LIN {X 0,Y 488.903,Z 502.562,A -85,B 0,C 180,E1 -6397.433,E2 -6397.433} C_VEL
LIN {X 0,Y 489.28,Z 495.024,A -85,B 0,C 180,E1 -6398.466,E2 -6398.466} C_VEL
LIN {X 0,Y 489.694,Z 485.882,A -85,B 0,C 180,E1 -6399.5,E2 -6399.5} C_VEL
LIN {X 0,Y 490.138,Z 475.738,A -85,B 0,C 180,E1 -6400.429,E2 -6400.429} C_VEL
LIN {X 0,Y 490.63,Z 464.492,A -85,B 0,C 180,E1 -6401.254,E2 -6401.254} C_VEL
LIN {X 0,Y 491.092,Z 452.788,A -85,B 0,C 180,E1 -6401.924,E2 -6401.924} C_VEL
LIN {X 0,Y 491.44,Z 439.88,A -85,B 0,C 180,E1 -6402.465,E2 -6402.465} C_VEL
LIN {X 0,Y 491.704,Z 427.075,A -85,B 0,C 180,E1 -6402.826,E2 -6402.826} C_VEL
LIN {X 0,Y 491.912,Z 400.381,A -85,B 0,C 180,E1 -6403.231,E2 -6403.231} C_VEL
LIN {X 0,Y 492.066,Z 328.64,A -85,B 0,C 180,E1 -6404.235,E2 -6404.235} C_VEL
LIN {X 0,Y 489.749,Z 314.502,A -85,B 0,C 180,E1 -6404.544,E2 -6404.544} C_VEL
LIN {X 0,Y 490.353,Z 294.957,A -85,B 0,C 180,E1 -6407.516,E2 -6407.516} C_VEL
LIN {X 0,Y 491.06,Z 277.065,A -85,B 0,C 180,E1 -6410.307,E2 -6410.307} C_VEL
LIN {X 0,Y 491.763,Z 261.922,A -85,B 0,C 180,E1 -6412.697,E2 -6412.697} C_VEL
LIN {X 0,Y 489.503,Z 250.936,A -85,B 0,C 180,E1 -6414.605,E2 -6414.605} C_VEL
LIN {X 0,Y 488.736,Z 247.293,A -85,B 0,C 180,E1 -6415.295,E2 -6415.295} C_VEL
LIN {X 0,Y 488.749,Z 247.222,A -85,B 0,C 180,E1 -6417.396,E2 -6417.396} C_VEL
LIN {X 0,Y 488.712,Z 247.228,A -85,B 0,C 180,E1 -6420.362,E2 -6420.362} C_VEL
LIN {X 0,Y 488.736,Z 247.219,A -85,B 0,C 180,E1 -6423.483,E2 -6423.483} C_VEL
LIN {X 0,Y 488.683,Z 247.236,A -85,B 0,C 180,E1 -6426.354,E2 -6426.354} C_VEL
LIN {X 0,Y 488.701,Z 247.239,A -85,B 0,C 180,E1 -6429.253,E2 -6429.253} C_VEL
LIN {X 0,Y 488.724,Z 247.232,A -85,B 0,C 180,E1 -6431.601,E2 -6431.601} C_VEL
LIN {X 0,Y 488.711,Z 247.231,A -85,B 0,C 180,E1 -6434.8,E2 -6434.8} C_VEL
LIN {X 0,Y 488.689,Z 247.237,A -85,B 0,C 180,E1 -6437.474,E2 -6437.474} C_VEL
LIN {X 0,Y 488.731,Z 247.22,A -85,B 0,C 180,E1 -6439.676,E2 -6439.676} C_VEL
LIN {X 0,Y 488.68,Z 247.238,A -85,B 0,C 180,E1 -6442.841,E2 -6442.841} C_VEL
LIN {X 0,Y 488.731,Z 247.217,A -85,B 0,C 180,E1 -6445.887,E2 -6445.887} C_VEL
LIN {X 0,Y 488.693,Z 247.235,A -85,B 0,C 180,E1 -6448.82,E2 -6448.82} C_VEL
LIN {X 0,Y 488.741,Z 247.224,A -85,B 0,C 180,E1 -6451.671,E2 -6451.671} C_VEL
LIN {X 0,Y 488.743,Z 247.229,A -85,B 0,C 180,E1 -6454.444,E2 -6454.444} C_VEL
LIN {X 0,Y 488.719,Z 247.233,A -85,B 0,C 180,E1 -6457.153,E2 -6457.153} C_VEL
LIN {X 0,Y 488.719,Z 247.226,A -85,B 0,C 180,E1 -6459.81,E2 -6459.81} C_VEL
LIN {X 0,Y 488.729,Z 247.231,A -85,B 0,C 180,E1 -6462.423,E2 -6462.423} C_VEL
LIN {X 0,Y 488.756,Z 247.226,A -85,B 0,C 180,E1 -6464.999,E2 -6464.999} C_VEL
LIN {X 0,Y 488.799,Z 247.224,A -85,B 0,C 180,E1 -6468.387,E2 -6468.387} C_VEL
LIN {X 0,Y 488.811,Z 247.217,A -85,B 0,C 180,E1 -6471.733,E2 -6471.733} C_VEL
LIN {X 0,Y 488.848,Z 247.216,A -85,B 0,C 180,E1 -6474.224,E2 -6474.224} C_VEL
LIN {X 0,Y 488.954,Z 247.199,A -85,B 0,C 180,E1 -6477.528,E2 -6477.528} C_VEL
LIN {X 0,Y 488.948,Z 247.201,A -85,B 0,C 180,E1 -6480.823,E2 -6480.823} C_VEL
LIN {X 0,Y 488.954,Z 247.206,A -85,B 0,C 180,E1 -6482.471,E2 -6482.471} C_VEL
LIN {X 0,Y 488.848,Z 247.211,A -85,B 0,C 180,E1 -6485.776,E2 -6485.776} C_VEL
LIN {X 0,Y 488.81,Z 247.224,A -85,B 0,C 180,E1 -6488.266,E2 -6488.266} C_VEL
LIN {X 0,Y 488.798,Z 247.215,A -85,B 0,C 180,E1 -6491.612,E2 -6491.612} C_VEL
LIN {X 0,Y 488.755,Z 247.223,A -85,B 0,C 180,E1 -6495,E2 -6495} C_VEL
LIN {X 0,Y 488.748,Z 247.23,A -85,B 0,C 180,E1 -6498.442,E2 -6498.442} C_VEL
LIN {X 0,Y 488.7,Z 247.229,A -85,B 0,C 180,E1 -6501.071,E2 -6501.071} C_VEL
LIN {X 0,Y 488.687,Z 247.237,A -85,B 0,C 180,E1 -6503.746,E2 -6503.746} C_VEL
LIN {X 0,Y 488.785,Z 247.221,A -85,B 0,C 180,E1 -6506.944,E2 -6506.944} C_VEL
LIN {X 0,Y 488.728,Z 247.221,A -85,B 0,C 180,E1 -6510.219,E2 -6510.219} C_VEL
LIN {X 0,Y 488.73,Z 247.23,A -85,B 0,C 180,E1 -6513.485,E2 -6513.485} C_VEL
LIN {X 0,Y 488.683,Z 247.226,A -85,B 0,C 180,E1 -6516.356,E2 -6516.356} C_VEL
LIN {X 0,Y 488.696,Z 247.234,A -85,B 0,C 180,E1 -6519.255,E2 -6519.255} C_VEL
LIN {X 0,Y 488.704,Z 247.233,A -85,B 0,C 180,E1 -6521.6,E2 -6521.6} C_VEL
LIN {X 0,Y 488.708,Z 247.231,A -85,B 0,C 180,E1 -6524.802,E2 -6524.802} C_VEL
LIN {X 0,Y 488.687,Z 247.219,A -85,B 0,C 180,E1 -6527.475,E2 -6527.475} C_VEL
LIN {X 0,Y 488.729,Z 247.221,A -85,B 0,C 180,E1 -6529.677,E2 -6529.677} C_VEL
LIN {X 0,Y 488.676,Z 247.233,A -85,B 0,C 180,E1 -6532.842,E2 -6532.842} C_VEL
LIN {X 0,Y 488.728,Z 247.234,A -85,B 0,C 180,E1 -6535.888,E2 -6535.888} C_VEL
LIN {X 0,Y 488.69,Z 247.226,A -85,B 0,C 180,E1 -6538.821,E2 -6538.821} C_VEL
LIN {X 0,Y 488.744,Z 247.222,A -85,B 0,C 180,E1 -6541.672,E2 -6541.672} C_VEL
LIN {X 0,Y 488.827,Z 247.449,A -85,B 0,C 180,E1 -6543.514,E2 -6543.514} C_VEL
LIN {X 0,Y 492.215,Z 262.595,A -85,B 0,C 180,E1 -6545.889,E2 -6545.889} C_VEL
LIN {X 0,Y 491.418,Z 281.498,A -85,B 0,C 180,E1 -6548.511,E2 -6548.511} C_VEL
LIN {X 0,Y 490.752,Z 296.315,A -85,B 0,C 180,E1 -6550.517,E2 -6550.517} C_VEL
LIN {X 0,Y 493.032,Z 311.538,A -85,B 0,C 180,E1 -6550.862,E2 -6550.862} C_VEL
LIN {X 0,Y 491.912,Z 432.787,A -85,B 0,C 180,E1 -6552.729,E2 -6552.729} C_VEL
LIN {X 0,Y 491.559,Z 447.226,A -85,B 0,C 180,E1 -6553.118,E2 -6553.118} C_VEL
LIN {X 0,Y 491.218,Z 460.741,A -85,B 0,C 180,E1 -6553.648,E2 -6553.648} C_VEL
LIN {X 0,Y 490.753,Z 473.693,A -85,B 0,C 180,E1 -6554.318,E2 -6554.318} C_VEL
LIN {X 0,Y 490.2,Z 486.396,A -85,B 0,C 180,E1 -6555.151,E2 -6555.151} C_VEL
LIN {X 0,Y 489.749,Z 497.984,A -85,B 0,C 180,E1 -6556.092,E2 -6556.092} C_VEL
LIN {X 0,Y 489.324,Z 508.613,A -85,B 0,C 180,E1 -6557.137,E2 -6557.137} C_VEL
LIN {X 0,Y 488.899,Z 519.163,A -85,B 0,C 180,E1 -6558.39,E2 -6558.39} C_VEL
LIN {X 0,Y 488.56,Z 527.847,A -85,B 0,C 180,E1 -6559.641,E2 -6559.641} C_VEL
LIN {X 0,Y 488.293,Z 536.116,A -85,B 0,C 180,E1 -6561.099,E2 -6561.099} C_VEL
LIN {X 0,Y 488.082,Z 542.76,A -85,B 0,C 180,E1 -6562.554,E2 -6562.554} C_VEL
LIN {X 0,Y 487.986,Z 547.46,A -85,B 0,C 180,E1 -6563.83,E2 -6563.83} C_VEL
LIN {X 0,Y 487.959,Z 550.963,A -85,B 0,C 180,E1 -6565.043,E2 -6565.043} C_VEL
LIN {X 0,Y 487.955,Z 554.478,A -85,B 0,C 180,E1 -6566.697,E2 -6566.697} C_VEL
LIN {X 0,Y 487.888,Z 556.557,A -85,B 0,C 180,E1 -6568.349,E2 -6568.349} C_VEL
LIN {X 0,Y 487.817,Z 557.248,A -85,B 0,C 180,E1 -6570,E2 -6570} C_VEL
LIN {X 0,Y 487.888,Z 556.557,A -85,B 0,C 180,E1 -6571.651,E2 -6571.651} C_VEL
LIN {X 0,Y 487.955,Z 554.479,A -85,B 0,C 180,E1 -6573.303,E2 -6573.303} C_VEL
LIN {X 0,Y 487.959,Z 550.963,A -85,B 0,C 180,E1 -6574.957,E2 -6574.957} C_VEL
LIN {X 0,Y 488.039,Z 545.903,A -85,B 0,C 180,E1 -6576.615,E2 -6576.615} C_VEL
LIN {X 0,Y 488.145,Z 540.999,A -85,B 0,C 180,E1 -6577.861,E2 -6577.861} C_VEL
LIN {X 0,Y 488.362,Z 533.898,A -85,B 0,C 180,E1 -6579.317,E2 -6579.317} C_VEL
LIN {X 0,Y 488.672,Z 525.079,A -85,B 0,C 180,E1 -6580.775,E2 -6580.775} C_VEL
LIN {X 0,Y 489.064,Z 515.126,A -85,B 0,C 180,E1 -6582.118,E2 -6582.118} C_VEL
LIN {X 0,Y 489.493,Z 503.551,A -85,B 0,C 180,E1 -6583.386,E2 -6583.386} C_VEL
LIN {X 0,Y 489.979,Z 491.858,A -85,B 0,C 180,E1 -6584.431,E2 -6584.431} C_VEL
LIN {X 0,Y 490.563,Z 478.879,A -85,B 0,C 180,E1 -6585.369,E2 -6585.369} C_VEL
LIN {X 0,Y 491.012,Z 465.403,A -85,B 0,C 180,E1 -6586.141,E2 -6586.141} C_VEL
LIN {X 0,Y 491.441,Z 451.989,A -85,B 0,C 180,E1 -6586.726,E2 -6586.726} C_VEL
LIN {X 0,Y 491.83,Z 437.712,A -85,B 0,C 180,E1 -6587.167,E2 -6587.167} C_VEL
LIN {X 0,Y 492.106,Z 421.126,A -85,B 0,C 180,E1 -6587.479,E2 -6587.479} C_VEL
LIN {X 0,Y 492.925,Z 309.57,A -85,B 0,C 180,E1 -6589.198,E2 -6589.198} C_VEL
LIN {X 0,Y 490.821,Z 296.434,A -85,B 0,C 180,E1 -6589.499,E2 -6589.499} C_VEL
LIN {X 0,Y 491.855,Z 273.118,A -85,B 0,C 180,E1 -6592.693,E2 -6592.693} C_VEL
LIN {X 0,Y 492.316,Z 262.77,A -85,B 0,C 180,E1 -6594.143,E2 -6594.143} C_VEL
LIN {X 0,Y 488.994,Z 248.173,A -85,B 0,C 180,E1 -6596.458,E2 -6596.458} C_VEL
LIN {X 0,Y 488.803,Z 247.293,A -85,B 0,C 180,E1 -6596.659,E2 -6596.659} C_VEL
LIN {X 0,Y 488.722,Z 247.228,A -85,B 0,C 180,E1 -6599.27,E2 -6599.27} C_VEL
LIN {X 0,Y 488.702,Z 247.223,A -85,B 0,C 180,E1 -6602.147,E2 -6602.147} C_VEL
LIN {X 0,Y 488.715,Z 247.227,A -85,B 0,C 180,E1 -6605.115,E2 -6605.115} C_VEL
LIN {X 0,Y 488.677,Z 247.234,A -85,B 0,C 180,E1 -6608.2,E2 -6608.2} C_VEL
LIN {X 0,Y 488.715,Z 247.232,A -85,B 0,C 180,E1 -6610.344,E2 -6610.344} C_VEL
LIN {X 0,Y 488.742,Z 247.228,A -85,B 0,C 180,E1 -6612.831,E2 -6612.831} C_VEL
LIN {X 0,Y 488.695,Z 247.235,A -85,B 0,C 180,E1 -6615.976,E2 -6615.976} C_VEL
LIN {X 0,Y 488.704,Z 247.228,A -85,B 0,C 180,E1 -6618.584,E2 -6618.584} C_VEL
LIN {X 0,Y 488.7,Z 247.233,A -85,B 0,C 180,E1 -6620.947,E2 -6620.947} C_VEL
LIN {X 0,Y 488.68,Z 247.231,A -85,B 0,C 180,E1 -6623.868,E2 -6623.868} C_VEL
LIN {X 0,Y 488.734,Z 247.228,A -85,B 0,C 180,E1 -6626.877,E2 -6626.877} C_VEL
LIN {X 0,Y 488.728,Z 247.223,A -85,B 0,C 180,E1 -6629.781,E2 -6629.781} C_VEL
LIN {X 0,Y 488.786,Z 247.22,A -85,B 0,C 180,E1 -6633.056,E2 -6633.056} C_VEL
LIN {X 0,Y 488.688,Z 247.237,A -85,B 0,C 180,E1 -6636.254,E2 -6636.254} C_VEL
LIN {X 0,Y 488.739,Z 247.225,A -85,B 0,C 180,E1 -6639.176,E2 -6639.176} C_VEL
LIN {X 0,Y 488.728,Z 247.228,A -85,B 0,C 180,E1 -6642.423,E2 -6642.423} C_VEL
LIN {X 0,Y 488.755,Z 247.223,A -85,B 0,C 180,E1 -6645,E2 -6645} C_VEL
LIN {X 0,Y 488.798,Z 247.217,A -85,B 0,C 180,E1 -6648.388,E2 -6648.388} C_VEL
LIN {X 0,Y 488.811,Z 247.22,A -85,B 0,C 180,E1 -6651.734,E2 -6651.734} C_VEL
LIN {X 0,Y 488.849,Z 247.214,A -85,B 0,C 180,E1 -6654.224,E2 -6654.224} C_VEL
LIN {X 0,Y 488.955,Z 247.202,A -85,B 0,C 180,E1 -6657.529,E2 -6657.529} C_VEL
LIN {X 0,Y 488.948,Z 247.201,A -85,B 0,C 180,E1 -6660.824,E2 -6660.824} C_VEL
LIN {X 0,Y 488.955,Z 247.195,A -85,B 0,C 180,E1 -6662.472,E2 -6662.472} C_VEL
LIN {X 0,Y 488.849,Z 247.214,A -85,B 0,C 180,E1 -6665.776,E2 -6665.776} C_VEL
LIN {X 0,Y 488.811,Z 247.217,A -85,B 0,C 180,E1 -6668.267,E2 -6668.267} C_VEL
LIN {X 0,Y 488.799,Z 247.221,A -85,B 0,C 180,E1 -6671.613,E2 -6671.613} C_VEL
LIN {X 0,Y 488.756,Z 247.228,A -85,B 0,C 180,E1 -6675.001,E2 -6675.001} C_VEL
LIN {X 0,Y 488.75,Z 247.226,A -85,B 0,C 180,E1 -6678.443,E2 -6678.443} C_VEL
LIN {X 0,Y 488.702,Z 247.235,A -85,B 0,C 180,E1 -6681.071,E2 -6681.071} C_VEL
LIN {X 0,Y 488.688,Z 247.232,A -85,B 0,C 180,E1 -6683.746,E2 -6683.746} C_VEL
LIN {X 0,Y 488.788,Z 247.226,A -85,B 0,C 180,E1 -6686.944,E2 -6686.944} C_VEL
LIN {X 0,Y 488.706,Z 247.226,A -85,B 0,C 180,E1 -6690.364,E2 -6690.364} C_VEL
LIN {X 0,Y 488.733,Z 247.226,A -85,B 0,C 180,E1 -6693.485,E2 -6693.485} C_VEL
LIN {X 0,Y 488.687,Z 247.231,A -85,B 0,C 180,E1 -6696.356,E2 -6696.356} C_VEL
LIN {X 0,Y 488.699,Z 247.228,A -85,B 0,C 180,E1 -6699.255,E2 -6699.255} C_VEL
LIN {X 0,Y 488.706,Z 247.232,A -85,B 0,C 180,E1 -6701.601,E2 -6701.601} C_VEL
LIN {X 0,Y 488.711,Z 247.232,A -85,B 0,C 180,E1 -6704.802,E2 -6704.802} C_VEL
LIN {X 0,Y 488.695,Z 247.23,A -85,B 0,C 180,E1 -6707.476,E2 -6707.476} C_VEL
LIN {X 0,Y 488.733,Z 247.228,A -85,B 0,C 180,E1 -6709.677,E2 -6709.677} C_VEL
LIN {X 0,Y 488.68,Z 247.229,A -85,B 0,C 180,E1 -6712.842,E2 -6712.842} C_VEL
LIN {X 0,Y 488.725,Z 247.221,A -85,B 0,C 180,E1 -6715.887,E2 -6715.887} C_VEL
LIN {X 0,Y 488.693,Z 247.228,A -85,B 0,C 180,E1 -6718.821,E2 -6718.821} C_VEL
LIN {X 0,Y 488.778,Z 247.428,A -85,B 0,C 180,E1 -6720.734,E2 -6720.734} C_VEL
LIN {X 0,Y 491.593,Z 260.102,A -85,B 0,C 180,E1 -6723.006,E2 -6723.006} C_VEL
LIN {X 0,Y 491.75,Z 264.568,A -85,B 0,C 180,E1 -6723.742,E2 -6723.742} C_VEL
LIN {X 0,Y 490.981,Z 268.147,A -85,B 0,C 180,E1 -6724.282,E2 -6724.282} C_VEL
LIN {X 0,Y 484.825,Z 280.462,A -85,B 0,C 180,E1 -6725.965,E2 -6725.965} C_VEL
LIN {X 0,Y 484.023,Z 284.083,A -85,B 0,C 180,E1 -6726.513,E2 -6726.513} C_VEL
LIN {X 0,Y 483.131,Z 304.815,A -85,B 0,C 180,E1 -6729.789,E2 -6729.789} C_VEL
LIN {X 0,Y 482.872,Z 314.366,A -85,B 0,C 180,E1 -6731.245,E2 -6731.245} C_VEL
LIN {X 0,Y 485.567,Z 331.287,A -85,B 0,C 180,E1 -6731.618,E2 -6731.618} C_VEL
LIN {X 0,Y 485.017,Z 426.075,A -85,B 0,C 180,E1 -6732.982,E2 -6732.982} C_VEL
LIN {X 0,Y 484.736,Z 438.363,A -85,B 0,C 180,E1 -6733.317,E2 -6733.317} C_VEL
LIN {X 0,Y 484.389,Z 451.485,A -85,B 0,C 180,E1 -6733.854,E2 -6733.854} C_VEL
LIN {X 0,Y 483.889,Z 463.426,A -85,B 0,C 180,E1 -6734.522,E2 -6734.522} C_VEL
LIN {X 0,Y 483.271,Z 474.991,A -85,B 0,C 180,E1 -6735.364,E2 -6735.364} C_VEL
LIN {X 0,Y 482.783,Z 485.373,A -85,B 0,C 180,E1 -6736.317,E2 -6736.317} C_VEL
LIN {X 0,Y 482.29,Z 494.732,A -85,B 0,C 180,E1 -6737.374,E2 -6737.374} C_VEL
LIN {X 0,Y 481.87,Z 503.739,A -85,B 0,C 180,E1 -6738.645,E2 -6738.645} C_VEL
LIN {X 0,Y 481.459,Z 510.996,A -85,B 0,C 180,E1 -6739.912,E2 -6739.912} C_VEL
LIN {X 0,Y 481.222,Z 516.822,A -85,B 0,C 180,E1 -6741.179,E2 -6741.179} C_VEL
LIN {X 0,Y 481.047,Z 521.433,A -85,B 0,C 180,E1 -6742.444,E2 -6742.444} C_VEL
LIN {X 0,Y 480.969,Z 524.542,A -85,B 0,C 180,E1 -6743.534,E2 -6743.534} C_VEL
LIN {X 0,Y 480.847,Z 527.539,A -85,B 0,C 180,E1 -6744.969,E2 -6744.969} C_VEL
LIN {X 0,Y 480.882,Z 529.583,A -85,B 0,C 180,E1 -6746.649,E2 -6746.649} C_VEL
LIN {X 0,Y 480.822,Z 530.056,A -85,B 0,C 180,E1 -6748.325,E2 -6748.325} C_VEL
LIN {X 0,Y 480.749,Z 529.064,A -85,B 0,C 180,E1 -6750,E2 -6750} C_VEL
LIN {X 0,Y 480.768,Z 527.997,A -85,B 0,C 180,E1 -6750.838,E2 -6750.838} C_VEL
LIN {X 0,Y 480.945,Z 524.621,A -85,B 0,C 180,E1 -6752.512,E2 -6752.512} C_VEL
LIN {X 0,Y 481.12,Z 520.982,A -85,B 0,C 180,E1 -6753.769,E2 -6753.769} C_VEL
LIN {X 0,Y 481.353,Z 516.273,A -85,B 0,C 180,E1 -6755.026,E2 -6755.026} C_VEL
LIN {X 0,Y 481.437,Z 510.363,A -85,B 0,C 180,E1 -6756.285,E2 -6756.285} C_VEL
LIN {X 0,Y 481.895,Z 503.017,A -85,B 0,C 180,E1 -6757.542,E2 -6757.542} C_VEL
LIN {X 0,Y 482.277,Z 495.538,A -85,B 0,C 180,E1 -6758.59,E2 -6758.59} C_VEL
LIN {X 0,Y 482.733,Z 486.492,A -85,B 0,C 180,E1 -6759.638,E2 -6759.638} C_VEL
LIN {X 0,Y 483.213,Z 476.447,A -85,B 0,C 180,E1 -6760.581,E2 -6760.581} C_VEL
LIN {X 0,Y 483.647,Z 466.885,A -85,B 0,C 180,E1 -6761.313,E2 -6761.313} C_VEL
LIN {X 0,Y 484.165,Z 454.778,A -85,B 0,C 180,E1 -6762.044,E2 -6762.044} C_VEL
LIN {X 0,Y 484.546,Z 442.05,A -85,B 0,C 180,E1 -6762.619,E2 -6762.619} C_VEL
LIN {X 0,Y 484.873,Z 429.222,A -85,B 0,C 180,E1 -6763.01,E2 -6763.01} C_VEL
LIN {X 0,Y 485.049,Z 412.381,A -85,B 0,C 180,E1 -6763.298,E2 -6763.298} C_VEL
LIN {X 0,Y 485.331,Z 329.733,A -85,B 0,C 180,E1 -6764.465,E2 -6764.465} C_VEL
LIN {X 0,Y 482.819,Z 314.79,A -85,B 0,C 180,E1 -6764.784,E2 -6764.784} C_VEL
LIN {X 0,Y 482.782,Z 313.033,A -85,B 0,C 180,E1 -6764.974,E2 -6764.974} C_VEL
LIN {X 0,Y 483.571,Z 292.331,A -85,B 0,C 180,E1 -6768.208,E2 -6768.208} C_VEL
LIN {X 0,Y 484.466,Z 271.755,A -85,B 0,C 180,E1 -6771.473,E2 -6771.473} C_VEL
LIN {X 0,Y 484.882,Z 263.407,A -85,B 0,C 180,E1 -6772.812,E2 -6772.812} C_VEL
LIN {X 0,Y 482.586,Z 252.416,A -85,B 0,C 180,E1 -6774.751,E2 -6774.751} C_VEL
LIN {X 0,Y 481.699,Z 248.184,A -85,B 0,C 180,E1 -6775.554,E2 -6775.554} C_VEL
LIN {X 0,Y 481.703,Z 248.108,A -85,B 0,C 180,E1 -6777.831,E2 -6777.831} C_VEL
LIN {X 0,Y 481.648,Z 248.108,A -85,B 0,C 180,E1 -6780.71,E2 -6780.71} C_VEL
LIN {X 0,Y 481.698,Z 248.095,A -85,B 0,C 180,E1 -6783.732,E2 -6783.732} C_VEL
LIN {X 0,Y 481.626,Z 248.116,A -85,B 0,C 180,E1 -6786.746,E2 -6786.746} C_VEL
LIN {X 0,Y 481.677,Z 248.107,A -85,B 0,C 180,E1 -6789.939,E2 -6789.939} C_VEL
LIN {X 0,Y 481.666,Z 248.114,A -85,B 0,C 180,E1 -6793.296,E2 -6793.296} C_VEL
LIN {X 0,Y 481.657,Z 248.109,A -85,B 0,C 180,E1 -6795.64,E2 -6795.64} C_VEL
LIN {X 0,Y 481.654,Z 248.112,A -85,B 0,C 180,E1 -6798.957,E2 -6798.957} C_VEL
LIN {X 0,Y 481.654,Z 248.109,A -85,B 0,C 180,E1 -6801.992,E2 -6801.992} C_VEL
LIN {X 0,Y 481.69,Z 248.098,A -85,B 0,C 180,E1 -6805.317,E2 -6805.317} C_VEL
LIN {X 0,Y 481.644,Z 248.108,A -85,B 0,C 180,E1 -6808.311,E2 -6808.311} C_VEL
LIN {X 0,Y 481.701,Z 248.104,A -85,B 0,C 180,E1 -6811.218,E2 -6811.218} C_VEL
LIN {X 0,Y 481.696,Z 248.104,A -85,B 0,C 180,E1 -6814.042,E2 -6814.042} C_VEL
LIN {X 0,Y 481.669,Z 248.111,A -85,B 0,C 180,E1 -6816.811,E2 -6816.811} C_VEL
LIN {X 0,Y 481.69,Z 248.102,A -85,B 0,C 180,E1 -6819.502,E2 -6819.502} C_VEL
LIN {X 0,Y 481.702,Z 248.104,A -85,B 0,C 180,E1 -6822.158,E2 -6822.158} C_VEL
LIN {X 0,Y 481.736,Z 248.101,A -85,B 0,C 180,E1 -6824.775,E2 -6824.775} C_VEL
LIN {X 0,Y 481.744,Z 248.101,A -85,B 0,C 180,E1 -6828.215,E2 -6828.215} C_VEL
LIN {X 0,Y 481.756,Z 248.095,A -85,B 0,C 180,E1 -6831.611,E2 -6831.611} C_VEL
LIN {X 0,Y 481.809,Z 248.092,A -85,B 0,C 180,E1 -6834.139,E2 -6834.139} C_VEL
LIN {X 0,Y 481.921,Z 248.076,A -85,B 0,C 180,E1 -6837.492,E2 -6837.492} C_VEL
LIN {X 0,Y 481.899,Z 248.079,A -85,B 0,C 180,E1 -6840.835,E2 -6840.835} C_VEL
LIN {X 0,Y 481.921,Z 248.083,A -85,B 0,C 180,E1 -6842.507,E2 -6842.507} C_VEL
LIN {X 0,Y 481.809,Z 248.088,A -85,B 0,C 180,E1 -6845.86,E2 -6845.86} C_VEL
LIN {X 0,Y 481.756,Z 248.104,A -85,B 0,C 180,E1 -6848.388,E2 -6848.388} C_VEL
LIN {X 0,Y 481.743,Z 248.095,A -85,B 0,C 180,E1 -6851.785,E2 -6851.785} C_VEL
LIN {X 0,Y 481.735,Z 248.096,A -85,B 0,C 180,E1 -6855.224,E2 -6855.224} C_VEL
LIN {X 0,Y 481.705,Z 248.104,A -85,B 0,C 180,E1 -6858.722,E2 -6858.722} C_VEL
LIN {X 0,Y 481.639,Z 248.109,A -85,B 0,C 180,E1 -6861.395,E2 -6861.395} C_VEL
LIN {X 0,Y 481.67,Z 248.111,A -85,B 0,C 180,E1 -6864.113,E2 -6864.113} C_VEL
LIN {X 0,Y 481.74,Z 248.099,A -85,B 0,C 180,E1 -6867.14,E2 -6867.14} C_VEL
LIN {X 0,Y 481.682,Z 248.101,A -85,B 0,C 180,E1 -6869.741,E2 -6869.741} C_VEL
LIN {X 0,Y 481.667,Z 248.108,A -85,B 0,C 180,E1 -6872.674,E2 -6872.674} C_VEL
LIN {X 0,Y 481.637,Z 248.113,A -85,B 0,C 180,E1 -6875.709,E2 -6875.709} C_VEL
LIN {X 0,Y 481.666,Z 248.108,A -85,B 0,C 180,E1 -6878.859,E2 -6878.859} C_VEL
LIN {X 0,Y 481.648,Z 248.109,A -85,B 0,C 180,E1 -6881.913,E2 -6881.913} C_VEL
LIN {X 0,Y 481.655,Z 248.11,A -85,B 0,C 180,E1 -6884.458,E2 -6884.458} C_VEL
LIN {X 0,Y 481.643,Z 248.092,A -85,B 0,C 180,E1 -6887.84,E2 -6887.84} C_VEL
LIN {X 0,Y 481.676,Z 248.107,A -85,B 0,C 180,E1 -6890.652,E2 -6890.652} C_VEL
LIN {X 0,Y 481.624,Z 248.107,A -85,B 0,C 180,E1 -6893.377,E2 -6893.377} C_VEL
LIN {X 0,Y 481.707,Z 248.105,A -85,B 0,C 180,E1 -6896.331,E2 -6896.331} C_VEL
LIN {X 0,Y 481.649,Z 248.109,A -85,B 0,C 180,E1 -6899.418,E2 -6899.418} C_VEL
LIN {X 0,Y 481.699,Z 248.102,A -85,B 0,C 180,E1 -6902.169,E2 -6902.169} C_VEL
LIN {X 0,Y 481.789,Z 248.313,A -85,B 0,C 180,E1 -6903.232,E2 -6903.232} C_VEL
LIN {X 0,Y 485.155,Z 262.825,A -85,B 0,C 180,E1 -6905.557,E2 -6905.557} C_VEL
LIN {X 0,Y 485.361,Z 266.39,A -85,B 0,C 180,E1 -6906.082,E2 -6906.082} C_VEL
LIN {X 0,Y 484.19,Z 288.433,A -85,B 0,C 180,E1 -6909.169,E2 -6909.169} C_VEL
LIN {X 0,Y 483.873,Z 296.527,A -85,B 0,C 180,E1 -6910.266,E2 -6910.266} C_VEL
LIN {X 0,Y 486.26,Z 312.164,A -85,B 0,C 180,E1 -6910.622,E2 -6910.622} C_VEL
LIN {X 0,Y 485.075,Z 432.499,A -85,B 0,C 180,E1 -6912.505,E2 -6912.505} C_VEL
LIN {X 0,Y 484.706,Z 446.985,A -85,B 0,C 180,E1 -6912.899,E2 -6912.899} C_VEL
LIN {X 0,Y 484.35,Z 460.351,A -85,B 0,C 180,E1 -6913.428,E2 -6913.428} C_VEL
LIN {X 0,Y 483.863,Z 473.042,A -85,B 0,C 180,E1 -6914.089,E2 -6914.089} C_VEL
LIN {X 0,Y 483.263,Z 485.836,A -85,B 0,C 180,E1 -6914.933,E2 -6914.933} C_VEL
LIN {X 0,Y 482.741,Z 497.493,A -85,B 0,C 180,E1 -6915.886,E2 -6915.886} C_VEL
LIN {X 0,Y 482.334,Z 508.179,A -85,B 0,C 180,E1 -6916.948,E2 -6916.948} C_VEL
LIN {X 0,Y 481.903,Z 518.78,A -85,B 0,C 180,E1 -6918.219,E2 -6918.219} C_VEL
LIN {X 0,Y 481.529,Z 527.504,A -85,B 0,C 180,E1 -6919.488,E2 -6919.488} C_VEL
LIN {X 0,Y 481.24,Z 535.815,A -85,B 0,C 180,E1 -6920.968,E2 -6920.968} C_VEL
LIN {X 0,Y 481.006,Z 542.489,A -85,B 0,C 180,E1 -6922.444,E2 -6922.444} C_VEL
LIN {X 0,Y 480.924,Z 546.655,A -85,B 0,C 180,E1 -6923.576,E2 -6923.576} C_VEL
LIN {X 0,Y 480.888,Z 550.732,A -85,B 0,C 180,E1 -6924.97,E2 -6924.97} C_VEL
LIN {X 0,Y 480.878,Z 554.263,A -85,B 0,C 180,E1 -6926.649,E2 -6926.649} C_VEL
LIN {X 0,Y 480.789,Z 556.354,A -85,B 0,C 180,E1 -6928.325,E2 -6928.325} C_VEL
LIN {X 0,Y 480.741,Z 557.049,A -85,B 0,C 180,E1 -6930,E2 -6930} C_VEL
LIN {X 0,Y 480.789,Z 556.354,A -85,B 0,C 180,E1 -6931.675,E2 -6931.675} C_VEL
LIN {X 0,Y 480.878,Z 554.265,A -85,B 0,C 180,E1 -6933.351,E2 -6933.351} C_VEL
LIN {X 0,Y 480.889,Z 550.731,A -85,B 0,C 180,E1 -6935.031,E2 -6935.031} C_VEL
LIN {X 0,Y 480.959,Z 545.652,A -85,B 0,C 180,E1 -6936.713,E2 -6936.713} C_VEL
LIN {X 0,Y 481.075,Z 540.729,A -85,B 0,C 180,E1 -6937.977,E2 -6937.977} C_VEL
LIN {X 0,Y 481.305,Z 533.61,A -85,B 0,C 180,E1 -6939.455,E2 -6939.455} C_VEL
LIN {X 0,Y 481.655,Z 524.775,A -85,B 0,C 180,E1 -6940.934,E2 -6940.934} C_VEL
LIN {X 0,Y 482.022,Z 515.572,A -85,B 0,C 180,E1 -6942.198,E2 -6942.198} C_VEL
LIN {X 0,Y 482.417,Z 505.296,A -85,B 0,C 180,E1 -6943.372,E2 -6943.372} C_VEL
LIN {X 0,Y 482.949,Z 494.064,A -85,B 0,C 180,E1 -6944.43,E2 -6944.43} C_VEL
LIN {X 0,Y 483.533,Z 481.647,A -85,B 0,C 180,E1 -6945.382,E2 -6945.382} C_VEL
LIN {X 0,Y 484.06,Z 468.631,A -85,B 0,C 180,E1 -6946.179,E2 -6946.179} C_VEL
LIN {X 0,Y 484.535,Z 455.487,A -85,B 0,C 180,E1 -6946.803,E2 -6946.803} C_VEL
LIN {X 0,Y 484.923,Z 440.828,A -85,B 0,C 180,E1 -6947.311,E2 -6947.311} C_VEL
LIN {X 0,Y 485.22,Z 426.625,A -85,B 0,C 180,E1 -6947.626,E2 -6947.626} C_VEL
LIN {X 0,Y 486.279,Z 311,A -85,B 0,C 180,E1 -6949.433,E2 -6949.433} C_VEL
LIN {X 0,Y 483.943,Z 296.431,A -85,B 0,C 180,E1 -6949.783,E2 -6949.783} C_VEL
LIN {X 0,Y 485.008,Z 274.754,A -85,B 0,C 180,E1 -6952.806,E2 -6952.806} C_VEL
LIN {X 0,Y 485.521,Z 264.759,A -85,B 0,C 180,E1 -6954.226,E2 -6954.226} C_VEL
LIN {X 0,Y 482.904,Z 252.943,A -85,B 0,C 180,E1 -6956.119,E2 -6956.119} C_VEL
LIN {X 0,Y 481.762,Z 248.221,A -85,B 0,C 180,E1 -6956.928,E2 -6956.928} C_VEL
LIN {X 0,Y 481.678,Z 248.109,A -85,B 0,C 180,E1 -6959.741,E2 -6959.741} C_VEL
LIN {X 0,Y 481.67,Z 248.102,A -85,B 0,C 180,E1 -6962.674,E2 -6962.674} C_VEL
LIN {X 0,Y 481.634,Z 248.104,A -85,B 0,C 180,E1 -6965.709,E2 -6965.709} C_VEL
LIN {X 0,Y 481.667,Z 248.112,A -85,B 0,C 180,E1 -6968.859,E2 -6968.859} C_VEL
LIN {X 0,Y 481.671,Z 248.112,A -85,B 0,C 180,E1 -6972.157,E2 -6972.157} C_VEL
LIN {X 0,Y 481.656,Z 248.109,A -85,B 0,C 180,E1 -6974.457,E2 -6974.457} C_VEL
LIN {X 0,Y 481.643,Z 248.114,A -85,B 0,C 180,E1 -6977.839,E2 -6977.839} C_VEL
LIN {X 0,Y 481.676,Z 248.11,A -85,B 0,C 180,E1 -6980.651,E2 -6980.651} C_VEL
LIN {X 0,Y 481.626,Z 248.108,A -85,B 0,C 180,E1 -6983.375,E2 -6983.375} C_VEL
LIN {X 0,Y 481.704,Z 248.108,A -85,B 0,C 180,E1 -6986.33,E2 -6986.33} C_VEL
LIN {X 0,Y 481.653,Z 248.105,A -85,B 0,C 180,E1 -6989.415,E2 -6989.415} C_VEL
LIN {X 0,Y 481.695,Z 248.108,A -85,B 0,C 180,E1 -6992.168,E2 -6992.168} C_VEL
LIN {X 0,Y 481.712,Z 248.1,A -85,B 0,C 180,E1 -6994.97,E2 -6994.97} C_VEL
LIN {X 0,Y 481.647,Z 248.116,A -85,B 0,C 180,E1 -6997.705,E2 -6997.705} C_VEL
LIN {X 0,Y 481.699,Z 248.105,A -85,B 0,C 180,E1 -7000.393,E2 -7000.393} C_VEL
LIN {X 0,Y 481.685,Z 248.104,A -85,B 0,C 180,E1 -7003.034,E2 -7003.034} C_VEL
LIN {X 0,Y 481.684,Z 248.11,A -85,B 0,C 180,E1 -7005.639,E2 -7005.639} C_VEL
LIN {X 0,Y 481.744,Z 248.097,A -85,B 0,C 180,E1 -7008.215,E2 -7008.215} C_VEL
LIN {X 0,Y 481.756,Z 248.101,A -85,B 0,C 180,E1 -7011.612,E2 -7011.612} C_VEL
LIN {X 0,Y 481.81,Z 248.092,A -85,B 0,C 180,E1 -7014.14,E2 -7014.14} C_VEL
LIN {X 0,Y 481.921,Z 248.078,A -85,B 0,C 180,E1 -7017.493,E2 -7017.493} C_VEL
LIN {X 0,Y 481.899,Z 248.079,A -85,B 0,C 180,E1 -7020.836,E2 -7020.836} C_VEL
LIN {X 0,Y 481.922,Z 248.071,A -85,B 0,C 180,E1 -7022.508,E2 -7022.508} C_VEL
LIN {X 0,Y 481.81,Z 248.089,A -85,B 0,C 180,E1 -7025.861,E2 -7025.861} C_VEL
LIN {X 0,Y 481.757,Z 248.095,A -85,B 0,C 180,E1 -7028.389,E2 -7028.389} C_VEL
LIN {X 0,Y 481.744,Z 248.098,A -85,B 0,C 180,E1 -7031.785,E2 -7031.785} C_VEL
LIN {X 0,Y 481.737,Z 248.103,A -85,B 0,C 180,E1 -7035.225,E2 -7035.225} C_VEL
LIN {X 0,Y 481.707,Z 248.105,A -85,B 0,C 180,E1 -7038.722,E2 -7038.722} C_VEL
LIN {X 0,Y 481.641,Z 248.117,A -85,B 0,C 180,E1 -7041.395,E2 -7041.395} C_VEL
LIN {X 0,Y 481.672,Z 248.105,A -85,B 0,C 180,E1 -7044.114,E2 -7044.114} C_VEL
LIN {X 0,Y 481.743,Z 248.1,A -85,B 0,C 180,E1 -7047.14,E2 -7047.14} C_VEL
LIN {X 0,Y 481.675,Z 248.102,A -85,B 0,C 180,E1 -7049.742,E2 -7049.742} C_VEL
LIN {X 0,Y 481.67,Z 248.112,A -85,B 0,C 180,E1 -7052.675,E2 -7052.675} C_VEL
LIN {X 0,Y 481.64,Z 248.107,A -85,B 0,C 180,E1 -7055.71,E2 -7055.71} C_VEL
LIN {X 0,Y 481.669,Z 248.109,A -85,B 0,C 180,E1 -7058.86,E2 -7058.86} C_VEL
LIN {X 0,Y 481.651,Z 248.11,A -85,B 0,C 180,E1 -7061.914,E2 -7061.914} C_VEL
LIN {X 0,Y 481.659,Z 248.107,A -85,B 0,C 180,E1 -7064.458,E2 -7064.458} C_VEL
LIN {X 0,Y 481.654,Z 248.106,A -85,B 0,C 180,E1 -7067.841,E2 -7067.841} C_VEL
LIN {X 0,Y 481.68,Z 248.1,A -85,B 0,C 180,E1 -7070.652,E2 -7070.652} C_VEL
LIN {X 0,Y 481.628,Z 248.116,A -85,B 0,C 180,E1 -7073.377,E2 -7073.377} C_VEL
LIN {X 0,Y 481.678,Z 248.099,A -85,B 0,C 180,E1 -7076.328,E2 -7076.328} C_VEL
LIN {X 0,Y 481.651,Z 248.104,A -85,B 0,C 180,E1 -7079.418,E2 -7079.418} C_VEL
LIN {X 0,Y 481.733,Z 248.297,A -85,B 0,C 180,E1 -7080.441,E2 -7080.441} C_VEL
LIN {X 0,Y 484.632,Z 261.337,A -85,B 0,C 180,E1 -7082.819,E2 -7082.819} C_VEL
LIN {X 0,Y 484.911,Z 265.943,A -85,B 0,C 180,E1 -7083.597,E2 -7083.597} C_VEL
LIN {X 0,Y 484.023,Z 284.083,A -85,B 0,C 180,E1 -7086.513,E2 -7086.513} C_VEL
LIN {X 0,Y 483.233,Z 287.692,A -85,B 0,C 180,E1 -7087.059,E2 -7087.059} C_VEL
LIN {X 0,Y 477.084,Z 300.013,A -85,B 0,C 180,E1 -7088.769,E2 -7088.769} C_VEL
LIN {X 0,Y 476.264,Z 303.664,A -85,B 0,C 180,E1 -7089.322,E2 -7089.322} C_VEL
LIN {X 0,Y 475.914,Z 314.104,A -85,B 0,C 180,E1 -7090.948,E2 -7090.948} C_VEL
LIN {X 0,Y 477.652,Z 324.167,A -85,B 0,C 180,E1 -7091.198,E2 -7091.198} C_VEL
LIN {X 0,Y 478.83,Z 331.515,A -85,B 0,C 180,E1 -7091.354,E2 -7091.354} C_VEL
LIN {X 0,Y 478.26,Z 425.217,A -85,B 0,C 180,E1 -7092.711,E2 -7092.711} C_VEL
LIN {X 0,Y 477.927,Z 438.447,A -85,B 0,C 180,E1 -7093.069,E2 -7093.069} C_VEL
LIN {X 0,Y 477.582,Z 450.94,A -85,B 0,C 180,E1 -7093.584,E2 -7093.584} C_VEL
LIN {X 0,Y 477.031,Z 463.568,A -85,B 0,C 180,E1 -7094.293,E2 -7094.293} C_VEL
LIN {X 0,Y 476.413,Z 475.133,A -85,B 0,C 180,E1 -7095.149,E2 -7095.149} C_VEL
LIN {X 0,Y 475.865,Z 485.515,A -85,B 0,C 180,E1 -7096.114,E2 -7096.114} C_VEL
LIN {X 0,Y 475.328,Z 494.876,A -85,B 0,C 180,E1 -7097.186,E2 -7097.186} C_VEL
LIN {X 0,Y 474.924,Z 502.546,A -85,B 0,C 180,E1 -7098.26,E2 -7098.26} C_VEL
LIN {X 0,Y 474.512,Z 510.051,A -85,B 0,C 180,E1 -7099.547,E2 -7099.547} C_VEL
LIN {X 0,Y 474.167,Z 516.974,A -85,B 0,C 180,E1 -7101.047,E2 -7101.047} C_VEL
LIN {X 0,Y 473.985,Z 521.589,A -85,B 0,C 180,E1 -7102.331,E2 -7102.331} C_VEL
LIN {X 0,Y 473.876,Z 524.991,A -85,B 0,C 180,E1 -7103.555,E2 -7103.555} C_VEL
LIN {X 0,Y 473.778,Z 527.708,A -85,B 0,C 180,E1 -7104.894,E2 -7104.894} C_VEL
LIN {X 0,Y 473.807,Z 529.765,A -85,B 0,C 180,E1 -7106.599,E2 -7106.599} C_VEL
LIN {X 0,Y 473.725,Z 530.26,A -85,B 0,C 180,E1 -7108.3,E2 -7108.3} C_VEL
LIN {X 0,Y 473.675,Z 529.288,A -85,B 0,C 180,E1 -7110,E2 -7110} C_VEL
LIN {X 0,Y 473.697,Z 528.24,A -85,B 0,C 180,E1 -7110.85,E2 -7110.85} C_VEL
LIN {X 0,Y 473.862,Z 524.897,A -85,B 0,C 180,E1 -7112.55,E2 -7112.55} C_VEL
LIN {X 0,Y 474.045,Z 521.289,A -85,B 0,C 180,E1 -7113.825,E2 -7113.825} C_VEL
LIN {X 0,Y 474.281,Z 516.615,A -85,B 0,C 180,E1 -7115.101,E2 -7115.101} C_VEL
LIN {X 0,Y 474.414,Z 510.745,A -85,B 0,C 180,E1 -7116.379,E2 -7116.379} C_VEL
LIN {X 0,Y 474.877,Z 503.446,A -85,B 0,C 180,E1 -7117.654,E2 -7117.654} C_VEL
LIN {X 0,Y 475.289,Z 496.017,A -85,B 0,C 180,E1 -7118.717,E2 -7118.717} C_VEL
LIN {X 0,Y 475.782,Z 487.043,A -85,B 0,C 180,E1 -7119.78,E2 -7119.78} C_VEL
LIN {X 0,Y 476.283,Z 477.114,A -85,B 0,C 180,E1 -7120.736,E2 -7120.736} C_VEL
LIN {X 0,Y 476.812,Z 466.105,A -85,B 0,C 180,E1 -7121.585,E2 -7121.585} C_VEL
LIN {X 0,Y 477.389,Z 453.747,A -85,B 0,C 180,E1 -7122.325,E2 -7122.325} C_VEL
LIN {X 0,Y 477.738,Z 441.936,A -85,B 0,C 180,E1 -7122.856,E2 -7122.856} C_VEL
LIN {X 0,Y 478.071,Z 428.936,A -85,B 0,C 180,E1 -7123.252,E2 -7123.252} C_VEL
LIN {X 0,Y 478.244,Z 411.828,A -85,B 0,C 180,E1 -7123.545,E2 -7123.545} C_VEL
LIN {X 0,Y 478.523,Z 330.247,A -85,B 0,C 180,E1 -7124.713,E2 -7124.713} C_VEL
LIN {X 0,Y 475.872,Z 314.441,A -85,B 0,C 180,E1 -7125.06,E2 -7125.06} C_VEL
LIN {X 0,Y 475.895,Z 311.799,A -85,B 0,C 180,E1 -7125.416,E2 -7125.416} C_VEL
LIN {X 0,Y 476.81,Z 289.704,A -85,B 0,C 180,E1 -7128.921,E2 -7128.921} C_VEL
LIN {X 0,Y 477.746,Z 269.463,A -85,B 0,C 180,E1 -7132.187,E2 -7132.187} C_VEL
LIN {X 0,Y 478.016,Z 264.891,A -85,B 0,C 180,E1 -7132.93,E2 -7132.93} C_VEL
LIN {X 0,Y 475.407,Z 252.518,A -85,B 0,C 180,E1 -7135.151,E2 -7135.151} C_VEL
LIN {X 0,Y 474.672,Z 249.052,A -85,B 0,C 180,E1 -7135.833,E2 -7135.833} C_VEL
LIN {X 0,Y 474.648,Z 248.987,A -85,B 0,C 180,E1 -7138.282,E2 -7138.282} C_VEL
LIN {X 0,Y 474.601,Z 248.991,A -85,B 0,C 180,E1 -7141.217,E2 -7141.217} C_VEL
LIN {X 0,Y 474.633,Z 248.977,A -85,B 0,C 180,E1 -7144.24,E2 -7144.24} C_VEL
LIN {X 0,Y 474.59,Z 248.992,A -85,B 0,C 180,E1 -7147.383,E2 -7147.383} C_VEL
LIN {X 0,Y 474.627,Z 248.987,A -85,B 0,C 180,E1 -7149.647,E2 -7149.647} C_VEL
LIN {X 0,Y 474.635,Z 248.988,A -85,B 0,C 180,E1 -7152.931,E2 -7152.931} C_VEL
LIN {X 0,Y 474.608,Z 248.986,A -85,B 0,C 180,E1 -7155.894,E2 -7155.894} C_VEL
LIN {X 0,Y 474.625,Z 248.985,A -85,B 0,C 180,E1 -7159.04,E2 -7159.04} C_VEL
LIN {X 0,Y 474.608,Z 248.988,A -85,B 0,C 180,E1 -7161.703,E2 -7161.703} C_VEL
LIN {X 0,Y 474.627,Z 248.988,A -85,B 0,C 180,E1 -7164.725,E2 -7164.725} C_VEL
LIN {X 0,Y 474.634,Z 248.98,A -85,B 0,C 180,E1 -7167.787,E2 -7167.787} C_VEL
LIN {X 0,Y 474.627,Z 248.99,A -85,B 0,C 180,E1 -7170.882,E2 -7170.882} C_VEL
LIN {X 0,Y 474.655,Z 248.982,A -85,B 0,C 180,E1 -7173.628,E2 -7173.628} C_VEL
LIN {X 0,Y 474.63,Z 248.985,A -85,B 0,C 180,E1 -7176.641,E2 -7176.641} C_VEL
LIN {X 0,Y 474.649,Z 248.979,A -85,B 0,C 180,E1 -7180.089,E2 -7180.089} C_VEL
LIN {X 0,Y 474.645,Z 248.989,A -85,B 0,C 180,E1 -7182.774,E2 -7182.774} C_VEL
LIN {X 0,Y 474.643,Z 248.98,A -85,B 0,C 180,E1 -7185.42,E2 -7185.42} C_VEL
LIN {X 0,Y 474.697,Z 248.977,A -85,B 0,C 180,E1 -7188.037,E2 -7188.037} C_VEL
LIN {X 0,Y 474.721,Z 248.972,A -85,B 0,C 180,E1 -7191.486,E2 -7191.486} C_VEL
LIN {X 0,Y 474.772,Z 248.968,A -85,B 0,C 180,E1 -7194.052,E2 -7194.052} C_VEL
LIN {X 0,Y 474.888,Z 248.952,A -85,B 0,C 180,E1 -7197.455,E2 -7197.455} C_VEL
LIN {X 0,Y 474.904,Z 248.95,A -85,B 0,C 180,E1 -7200,E2 -7200} C_VEL
LIN {X 0,Y 474.887,Z 248.959,A -85,B 0,C 180,E1 -7202.544,E2 -7202.544} C_VEL
LIN {X 0,Y 474.772,Z 248.965,A -85,B 0,C 180,E1 -7205.947,E2 -7205.947} C_VEL
LIN {X 0,Y 474.721,Z 248.978,A -85,B 0,C 180,E1 -7208.513,E2 -7208.513} C_VEL
LIN {X 0,Y 474.696,Z 248.975,A -85,B 0,C 180,E1 -7211.962,E2 -7211.962} C_VEL
LIN {X 0,Y 474.692,Z 248.974,A -85,B 0,C 180,E1 -7215.456,E2 -7215.456} C_VEL
LIN {X 0,Y 474.658,Z 248.98,A -85,B 0,C 180,E1 -7219.01,E2 -7219.01} C_VEL
LIN {X 0,Y 474.583,Z 248.991,A -85,B 0,C 180,E1 -7221.729,E2 -7221.729} C_VEL
LIN {X 0,Y 474.652,Z 248.981,A -85,B 0,C 180,E1 -7224.493,E2 -7224.493} C_VEL
LIN {X 0,Y 474.692,Z 248.977,A -85,B 0,C 180,E1 -7227.339,E2 -7227.339} C_VEL
LIN {X 0,Y 474.604,Z 248.977,A -85,B 0,C 180,E1 -7230.812,E2 -7230.812} C_VEL
LIN {X 0,Y 474.633,Z 248.991,A -85,B 0,C 180,E1 -7233.984,E2 -7233.984} C_VEL
LIN {X 0,Y 474.569,Z 248.981,A -85,B 0,C 180,E1 -7236.9,E2 -7236.9} C_VEL
LIN {X 0,Y 474.623,Z 248.992,A -85,B 0,C 180,E1 -7239.648,E2 -7239.648} C_VEL
LIN {X 0,Y 474.61,Z 248.983,A -85,B 0,C 180,E1 -7242.935,E2 -7242.935} C_VEL
LIN {X 0,Y 474.604,Z 248.984,A -85,B 0,C 180,E1 -7245.896,E2 -7245.896} C_VEL
LIN {X 0,Y 474.624,Z 248.968,A -85,B 0,C 180,E1 -7249.041,E2 -7249.041} C_VEL
LIN {X 0,Y 474.606,Z 248.993,A -85,B 0,C 180,E1 -7251.705,E2 -7251.705} C_VEL
LIN {X 0,Y 474.621,Z 248.976,A -85,B 0,C 180,E1 -7254.726,E2 -7254.726} C_VEL
LIN {X 0,Y 474.634,Z 248.977,A -85,B 0,C 180,E1 -7257.788,E2 -7257.788} C_VEL
LIN {X 0,Y 474.622,Z 248.984,A -85,B 0,C 180,E1 -7260.885,E2 -7260.885} C_VEL
LIN {X 0,Y 474.729,Z 249.113,A -85,B 0,C 180,E1 -7262.921,E2 -7262.921} C_VEL
LIN {X 0,Y 478.391,Z 264.907,A -85,B 0,C 180,E1 -7265.503,E2 -7265.503} C_VEL
LIN {X 0,Y 478.44,Z 269.477,A -85,B 0,C 180,E1 -7266.175,E2 -7266.175} C_VEL
LIN {X 0,Y 477.272,Z 289.925,A -85,B 0,C 180,E1 -7269.079,E2 -7269.079} C_VEL
LIN {X 0,Y 477,Z 296.495,A -85,B 0,C 180,E1 -7269.99,E2 -7269.99} C_VEL
LIN {X 0,Y 479.486,Z 313.34,A -85,B 0,C 180,E1 -7270.386,E2 -7270.386} C_VEL
LIN {X 0,Y 478.256,Z 432.217,A -85,B 0,C 180,E1 -7272.274,E2 -7272.274} C_VEL
LIN {X 0,Y 477.856,Z 446.756,A -85,B 0,C 180,E1 -7272.673,E2 -7272.673} C_VEL
LIN {X 0,Y 477.46,Z 461,A -85,B 0,C 180,E1 -7273.251,E2 -7273.251} C_VEL
LIN {X 0,Y 476.902,Z 474.185,A -85,B 0,C 180,E1 -7273.96,E2 -7273.96} C_VEL
LIN {X 0,Y 476.273,Z 486.735,A -85,B 0,C 180,E1 -7274.816,E2 -7274.816} C_VEL
LIN {X 0,Y 475.731,Z 498.208,A -85,B 0,C 180,E1 -7275.783,E2 -7275.783} C_VEL
LIN {X 0,Y 475.262,Z 509.718,A -85,B 0,C 180,E1 -7276.967,E2 -7276.967} C_VEL
LIN {X 0,Y 474.796,Z 519.963,A -85,B 0,C 180,E1 -7278.257,E2 -7278.257} C_VEL
LIN {X 0,Y 474.429,Z 528.452,A -85,B 0,C 180,E1 -7279.545,E2 -7279.545} C_VEL
LIN {X 0,Y 474.138,Z 536.55,A -85,B 0,C 180,E1 -7281.046,E2 -7281.046} C_VEL
LIN {X 0,Y 473.929,Z 542.221,A -85,B 0,C 180,E1 -7282.33,E2 -7282.33} C_VEL
LIN {X 0,Y 473.848,Z 546.742,A -85,B 0,C 180,E1 -7283.579,E2 -7283.579} C_VEL
LIN {X 0,Y 473.816,Z 550.497,A -85,B 0,C 180,E1 -7284.894,E2 -7284.894} C_VEL
LIN {X 0,Y 473.785,Z 554.046,A -85,B 0,C 180,E1 -7286.598,E2 -7286.598} C_VEL
LIN {X 0,Y 473.695,Z 556.148,A -85,B 0,C 180,E1 -7288.3,E2 -7288.3} C_VEL
LIN {X 0,Y 473.668,Z 556.851,A -85,B 0,C 180,E1 -7290,E2 -7290} C_VEL
LIN {X 0,Y 473.695,Z 556.154,A -85,B 0,C 180,E1 -7291.7,E2 -7291.7} C_VEL
LIN {X 0,Y 473.785,Z 554.059,A -85,B 0,C 180,E1 -7293.402,E2 -7293.402} C_VEL
LIN {X 0,Y 473.818,Z 550.516,A -85,B 0,C 180,E1 -7295.106,E2 -7295.106} C_VEL
LIN {X 0,Y 473.889,Z 545.427,A -85,B 0,C 180,E1 -7296.814,E2 -7296.814} C_VEL
LIN {X 0,Y 474.019,Z 540.493,A -85,B 0,C 180,E1 -7298.097,E2 -7298.097} C_VEL
LIN {X 0,Y 474.226,Z 533.359,A -85,B 0,C 180,E1 -7299.597,E2 -7299.597} C_VEL
LIN {X 0,Y 474.637,Z 524.513,A -85,B 0,C 180,E1 -7301.098,E2 -7301.098} C_VEL
LIN {X 0,Y 475.088,Z 514.464,A -85,B 0,C 180,E1 -7302.488,E2 -7302.488} C_VEL
LIN {X 0,Y 475.525,Z 503.975,A -85,B 0,C 180,E1 -7303.678,E2 -7303.678} C_VEL
LIN {X 0,Y 476.061,Z 492.45,A -85,B 0,C 180,E1 -7304.753,E2 -7304.753} C_VEL
LIN {X 0,Y 476.709,Z 479.689,A -85,B 0,C 180,E1 -7305.717,E2 -7305.717} C_VEL
LIN {X 0,Y 477.225,Z 467.137,A -85,B 0,C 180,E1 -7306.476,E2 -7306.476} C_VEL
LIN {X 0,Y 477.71,Z 453.552,A -85,B 0,C 180,E1 -7307.112,E2 -7307.112} C_VEL
LIN {X 0,Y 478.194,Z 439.314,A -85,B 0,C 180,E1 -7307.59,E2 -7307.59} C_VEL
LIN {X 0,Y 478.495,Z 424.023,A -85,B 0,C 180,E1 -7307.91,E2 -7307.91} C_VEL
LIN {X 0,Y 479.491,Z 311.491,A -85,B 0,C 180,E1 -7309.696,E2 -7309.696} C_VEL
LIN {X 0,Y 477.068,Z 296.672,A -85,B 0,C 180,E1 -7310.057,E2 -7310.057} C_VEL
LIN {X 0,Y 478.171,Z 276.391,A -85,B 0,C 180,E1 -7312.922,E2 -7312.922} C_VEL
LIN {X 0,Y 478.633,Z 265.89,A -85,B 0,C 180,E1 -7314.443,E2 -7314.443} C_VEL
LIN {X 0,Y 475.329,Z 251.503,A -85,B 0,C 180,E1 -7316.805,E2 -7316.805} C_VEL
LIN {X 0,Y 474.708,Z 249.09,A -85,B 0,C 180,E1 -7317.251,E2 -7317.251} C_VEL
LIN {X 0,Y 474.604,Z 248.994,A -85,B 0,C 180,E1 -7320.23,E2 -7320.23} C_VEL
LIN {X 0,Y 474.641,Z 248.985,A -85,B 0,C 180,E1 -7323.22,E2 -7323.22} C_VEL
LIN {X 0,Y 474.586,Z 248.976,A -85,B 0,C 180,E1 -7326.323,E2 -7326.323} C_VEL
LIN {X 0,Y 474.624,Z 248.988,A -85,B 0,C 180,E1 -7329.647,E2 -7329.647} C_VEL
LIN {X 0,Y 474.649,Z 248.983,A -85,B 0,C 180,E1 -7332.93,E2 -7332.93} C_VEL
LIN {X 0,Y 474.605,Z 248.989,A -85,B 0,C 180,E1 -7335.895,E2 -7335.895} C_VEL
LIN {X 0,Y 474.623,Z 248.979,A -85,B 0,C 180,E1 -7339.04,E2 -7339.04} C_VEL
LIN {X 0,Y 474.606,Z 248.991,A -85,B 0,C 180,E1 -7341.704,E2 -7341.704} C_VEL
LIN {X 0,Y 474.625,Z 248.982,A -85,B 0,C 180,E1 -7344.726,E2 -7344.726} C_VEL
LIN {X 0,Y 474.633,Z 248.989,A -85,B 0,C 180,E1 -7347.788,E2 -7347.788} C_VEL
LIN {X 0,Y 474.625,Z 248.976,A -85,B 0,C 180,E1 -7350.883,E2 -7350.883} C_VEL
LIN {X 0,Y 474.655,Z 248.985,A -85,B 0,C 180,E1 -7353.628,E2 -7353.628} C_VEL
LIN {X 0,Y 474.63,Z 248.985,A -85,B 0,C 180,E1 -7356.641,E2 -7356.641} C_VEL
LIN {X 0,Y 474.648,Z 248.986,A -85,B 0,C 180,E1 -7360.089,E2 -7360.089} C_VEL
LIN {X 0,Y 474.645,Z 248.981,A -85,B 0,C 180,E1 -7362.774,E2 -7362.774} C_VEL
LIN {X 0,Y 474.642,Z 248.985,A -85,B 0,C 180,E1 -7365.421,E2 -7365.421} C_VEL
LIN {X 0,Y 474.697,Z 248.976,A -85,B 0,C 180,E1 -7368.038,E2 -7368.038} C_VEL
LIN {X 0,Y 474.722,Z 248.978,A -85,B 0,C 180,E1 -7371.487,E2 -7371.487} C_VEL
LIN {X 0,Y 474.772,Z 248.969,A -85,B 0,C 180,E1 -7374.053,E2 -7374.053} C_VEL
LIN {X 0,Y 474.888,Z 248.954,A -85,B 0,C 180,E1 -7377.456,E2 -7377.456} C_VEL
LIN {X 0,Y 474.905,Z 248.952,A -85,B 0,C 180,E1 -7380,E2 -7380} C_VEL
LIN {X 0,Y 474.888,Z 248.947,A -85,B 0,C 180,E1 -7382.545,E2 -7382.545} C_VEL
LIN {X 0,Y 474.773,Z 248.965,A -85,B 0,C 180,E1 -7385.948,E2 -7385.948} C_VEL
LIN {X 0,Y 474.722,Z 248.972,A -85,B 0,C 180,E1 -7388.514,E2 -7388.514} C_VEL
LIN {X 0,Y 474.698,Z 248.975,A -85,B 0,C 180,E1 -7391.963,E2 -7391.963} C_VEL
LIN {X 0,Y 474.694,Z 248.977,A -85,B 0,C 180,E1 -7395.456,E2 -7395.456} C_VEL
LIN {X 0,Y 474.66,Z 248.986,A -85,B 0,C 180,E1 -7399.011,E2 -7399.011} C_VEL
LIN {X 0,Y 474.584,Z 248.992,A -85,B 0,C 180,E1 -7401.73,E2 -7401.73} C_VEL
LIN {X 0,Y 474.654,Z 248.98,A -85,B 0,C 180,E1 -7404.494,E2 -7404.494} C_VEL
LIN {X 0,Y 474.677,Z 248.976,A -85,B 0,C 180,E1 -7407.335,E2 -7407.335} C_VEL
LIN {X 0,Y 474.602,Z 248.987,A -85,B 0,C 180,E1 -7410.811,E2 -7410.811} C_VEL
LIN {X 0,Y 474.635,Z 248.98,A -85,B 0,C 180,E1 -7413.985,E2 -7413.985} C_VEL
LIN {X 0,Y 474.573,Z 248.995,A -85,B 0,C 180,E1 -7416.901,E2 -7416.901} C_VEL
LIN {X 0,Y 474.616,Z 248.979,A -85,B 0,C 180,E1 -7419.647,E2 -7419.647} C_VEL
LIN {X 0,Y 474.613,Z 248.989,A -85,B 0,C 180,E1 -7422.935,E2 -7422.935} C_VEL
LIN {X 0,Y 474.615,Z 248.988,A -85,B 0,C 180,E1 -7425.897,E2 -7425.897} C_VEL
LIN {X 0,Y 474.633,Z 248.989,A -85,B 0,C 180,E1 -7429.041,E2 -7429.041} C_VEL
LIN {X 0,Y 474.61,Z 248.97,A -85,B 0,C 180,E1 -7431.705,E2 -7431.705} C_VEL
LIN {X 0,Y 474.624,Z 248.986,A -85,B 0,C 180,E1 -7434.726,E2 -7434.726} C_VEL
LIN {X 0,Y 474.636,Z 248.989,A -85,B 0,C 180,E1 -7437.788,E2 -7437.788} C_VEL
LIN {X 0,Y 474.667,Z 249.186,A -85,B 0,C 180,E1 -7440.143,E2 -7440.143} C_VEL
LIN {X 0,Y 477.739,Z 262.833,A -85,B 0,C 180,E1 -7442.674,E2 -7442.674} C_VEL
